LIN {X 0,Y 448.387,Z 731.206,A -85,B 0,C 180,E1 -8746.152,E2 -8746.152} C_VEL
LIN {X 0,Y 449.35,Z 719.289,A -85,B 0,C 180,E1 -8747.497,E2 -8747.497} C_VEL
LIN {X 0,Y 450.298,Z 706.862,A -85,B 0,C 180,E1 -8748.658,E2 -8748.658} C_VEL
LIN {X 0,Y 451.248,Z 693.533,A -85,B 0,C 180,E1 -8749.68,E2 -8749.68} C_VEL
LIN {X 0,Y 452.18,Z 678.745,A -85,B 0,C 180,E1 -8750.586,E2 -8750.586} C_VEL
LIN {X 0,Y 452.945,Z 663.719,A -85,B 0,C 180,E1 -8751.29,E2 -8751.29} C_VEL
LIN {X 0,Y 453.549,Z 648.187,A -85,B 0,C 180,E1 -8751.811,E2 -8751.811} C_VEL
LIN {X 0,Y 453.905,Z 632.846,A -85,B 0,C 180,E1 -8752.142,E2 -8752.142} C_VEL
LIN {X 0,Y 455.724,Z 493.743,A -85,B 0,C 180,E1 -8754.379,E2 -8754.379} C_VEL
LIN {X 0,Y 451.739,Z 464.618,A -85,B 0,C 180,E1 -8755.125,E2 -8755.125} C_VEL
LIN {X 0,Y 451.619,Z 462.28,A -85,B 0,C 180,E1 -8755.248,E2 -8755.248} C_VEL
LIN {X 0,Y 453.55,Z 429.737,A -85,B 0,C 180,E1 -8758.834,E2 -8758.834} C_VEL
LIN {X 0,Y 455.129,Z 405.936,A -85,B 0,C 180,E1 -8761.497,E2 -8761.497} C_VEL
LIN {X 0,Y 451.572,Z 392.919,A -85,B 0,C 180,E1 -8763.254,E2 -8763.254} C_VEL
LIN {X 0,Y 446.431,Z 375.769,A -85,B 0,C 180,E1 -8765.709,E2 -8765.709} C_VEL
LIN {X 0,Y 446.382,Z 375.506,A -85,B 0,C 180,E1 -8766.745,E2 -8766.745} C_VEL
LIN {X 0,Y 446.386,Z 375.51,A -85,B 0,C 180,E1 -8770.202,E2 -8770.202} C_VEL
LIN {X 0,Y 446.38,Z 375.506,A -85,B 0,C 180,E1 -8773.594,E2 -8773.594} C_VEL
LIN {X 0,Y 446.365,Z 375.494,A -85,B 0,C 180,E1 -8776.405,E2 -8776.405} C_VEL
LIN {X 0,Y 446.384,Z 375.498,A -85,B 0,C 180,E1 -8779.796,E2 -8779.796} C_VEL
LIN {X 0,Y 446.378,Z 375.492,A -85,B 0,C 180,E1 -8783.252,E2 -8783.252} C_VEL
LIN {X 0,Y 446.435,Z 375.484,A -85,B 0,C 180,E1 -8786.565,E2 -8786.565} C_VEL
LIN {X 0,Y 446.414,Z 375.501,A -85,B 0,C 180,E1 -8789.979,E2 -8789.979} C_VEL
LIN {X 0,Y 446.381,Z 375.507,A -85,B 0,C 180,E1 -8792.833,E2 -8792.833} C_VEL
LIN {X 0,Y 446.416,Z 375.492,A -85,B 0,C 180,E1 -8795.933,E2 -8795.933} C_VEL
LIN {X 0,Y 446.436,Z 375.494,A -85,B 0,C 180,E1 -8798.772,E2 -8798.772} C_VEL
LIN {X 0,Y 446.423,Z 375.497,A -85,B 0,C 180,E1 -8801.648,E2 -8801.648} C_VEL
LIN {X 0,Y 446.442,Z 375.491,A -85,B 0,C 180,E1 -8804.478,E2 -8804.478} C_VEL
LIN {X 0,Y 446.5,Z 375.489,A -85,B 0,C 180,E1 -8807.384,E2 -8807.384} C_VEL
LIN {X 0,Y 446.495,Z 375.484,A -85,B 0,C 180,E1 -8810.944,E2 -8810.944} C_VEL
LIN {X 0,Y 446.582,Z 375.478,A -85,B 0,C 180,E1 -8813.675,E2 -8813.675} C_VEL
LIN {X 0,Y 446.646,Z 375.469,A -85,B 0,C 180,E1 -8817.294,E2 -8817.294} C_VEL
LIN {X 0,Y 446.68,Z 375.466,A -85,B 0,C 180,E1 -8820,E2 -8820} C_VEL
LIN {X 0,Y 446.641,Z 375.472,A -85,B 0,C 180,E1 -8822.706,E2 -8822.706} C_VEL
LIN {X 0,Y 446.608,Z 375.47,A -85,B 0,C 180,E1 -8826.324,E2 -8826.324} C_VEL
LIN {X 0,Y 446.505,Z 375.49,A -85,B 0,C 180,E1 -8829.056,E2 -8829.056} C_VEL
LIN {X 0,Y 446.506,Z 375.484,A -85,B 0,C 180,E1 -8832.73,E2 -8832.73} C_VEL
LIN {X 0,Y 446.473,Z 375.486,A -85,B 0,C 180,E1 -8836.46,E2 -8836.46} C_VEL
LIN {X 0,Y 446.453,Z 375.494,A -85,B 0,C 180,E1 -8839.304,E2 -8839.304} C_VEL
LIN {X 0,Y 446.401,Z 375.497,A -85,B 0,C 180,E1 -8842.201,E2 -8842.201} C_VEL
LIN {X 0,Y 446.399,Z 375.496,A -85,B 0,C 180,E1 -8845.156,E2 -8845.156} C_VEL
LIN {X 0,Y 446.402,Z 375.504,A -85,B 0,C 180,E1 -8848.184,E2 -8848.184} C_VEL
LIN {X 0,Y 446.379,Z 375.507,A -85,B 0,C 180,E1 -8851.303,E2 -8851.303} C_VEL
LIN {X 0,Y 446.409,Z 375.507,A -85,B 0,C 180,E1 -8854.525,E2 -8854.525} C_VEL
LIN {X 0,Y 446.386,Z 375.486,A -85,B 0,C 180,E1 -8858.078,E2 -8858.078} C_VEL
LIN {X 0,Y 446.388,Z 375.497,A -85,B 0,C 180,E1 -8861.396,E2 -8861.396} C_VEL
LIN {X 0,Y 446.405,Z 375.504,A -85,B 0,C 180,E1 -8865.11,E2 -8865.11} C_VEL
LIN {X 0,Y 446.389,Z 375.51,A -85,B 0,C 180,E1 -8868.607,E2 -8868.607} C_VEL
LIN {X 0,Y 446.388,Z 375.506,A -85,B 0,C 180,E1 -8871.925,E2 -8871.925} C_VEL
LIN {X 0,Y 446.403,Z 375.73,A -85,B 0,C 180,E1 -8873.134,E2 -8873.134} C_VEL
LIN {X 0,Y 451.361,Z 391.214,A -85,B 0,C 180,E1 -8875.416,E2 -8875.416} C_VEL
LIN {X 0,Y 455.662,Z 406.671,A -85,B 0,C 180,E1 -8877.56,E2 -8877.56} C_VEL
LIN {X 0,Y 454.897,Z 422.239,A -85,B 0,C 180,E1 -8879.349,E2 -8879.349} C_VEL
LIN {X 0,Y 453.716,Z 445.705,A -85,B 0,C 180,E1 -8881.997,E2 -8881.997} C_VEL
LIN {X 0,Y 452.629,Z 471.656,A -85,B 0,C 180,E1 -8884.802,E2 -8884.802} C_VEL
LIN {X 0,Y 453.796,Z 479.214,A -85,B 0,C 180,E1 -8885.035,E2 -8885.035} C_VEL
LIN {X 0,Y 456.513,Z 495.836,A -85,B 0,C 180,E1 -8885.476,E2 -8885.476} C_VEL
LIN {X 0,Y 455.399,Z 574.472,A -85,B 0,C 180,E1 -8886.745,E2 -8886.745} C_VEL
LIN {X 0,Y 454.701,Z 580.317,A -85,B 0,C 180,E1 -8886.806,E2 -8886.806} C_VEL
LIN {X 0,Y 449.167,Z 599.361,A -85,B 0,C 180,E1 -8886.83,E2 -8886.83} C_VEL
LIN {X 0,Y 448.435,Z 605.208,A -85,B 0,C 180,E1 -8886.89,E2 -8886.89} C_VEL
LIN {X 0,Y 447.794,Z 641.594,A -85,B 0,C 180,E1 -8887.51,E2 -8887.51} C_VEL
LIN {X 0,Y 447.297,Z 656.597,A -85,B 0,C 180,E1 -8887.935,E2 -8887.935} C_VEL
LIN {X 0,Y 446.583,Z 670.422,A -85,B 0,C 180,E1 -8888.489,E2 -8888.489} C_VEL
LIN {X 0,Y 445.726,Z 684.345,A -85,B 0,C 180,E1 -8889.222,E2 -8889.222} C_VEL
LIN {X 0,Y 444.669,Z 698.114,A -85,B 0,C 180,E1 -8890.137,E2 -8890.137} C_VEL
LIN {X 0,Y 443.595,Z 712.023,A -85,B 0,C 180,E1 -8891.289,E2 -8891.289} C_VEL
LIN {X 0,Y 442.535,Z 724.573,A -85,B 0,C 180,E1 -8892.559,E2 -8892.559} C_VEL
LIN {X 0,Y 441.589,Z 735.099,A -85,B 0,C 180,E1 -8893.83,E2 -8893.83} C_VEL
LIN {X 0,Y 440.61,Z 746.313,A -85,B 0,C 180,E1 -8895.452,E2 -8895.452} C_VEL
LIN {X 0,Y 439.871,Z 755.606,A -85,B 0,C 180,E1 -8897.076,E2 -8897.076} C_VEL
LIN {X 0,Y 439.437,Z 762.344,A -85,B 0,C 180,E1 -8898.47,E2 -8898.47} C_VEL
LIN {X 0,Y 438.855,Z 769.757,A -85,B 0,C 180,E1 -8900.321,E2 -8900.321} C_VEL
LIN {X 0,Y 438.543,Z 775.645,A -85,B 0,C 180,E1 -8902.172,E2 -8902.172} C_VEL
LIN {X 0,Y 438.365,Z 779.494,A -85,B 0,C 180,E1 -8903.723,E2 -8903.723} C_VEL
LIN {X 0,Y 438.3,Z 782.66,A -85,B 0,C 180,E1 -8905.403,E2 -8905.403} C_VEL
LIN {X 0,Y 438.286,Z 785.001,A -85,B 0,C 180,E1 -8907.244,E2 -8907.244} C_VEL
LIN {X 0,Y 438.227,Z 786.195,A -85,B 0,C 180,E1 -8909.083,E2 -8909.083} C_VEL
LIN {X 0,Y 438.228,Z 786.212,A -85,B 0,C 180,E1 -8910.92,E2 -8910.92} C_VEL
LIN {X 0,Y 438.287,Z 785.081,A -85,B 0,C 180,E1 -8912.759,E2 -8912.759} C_VEL
LIN {X 0,Y 438.3,Z 782.802,A -85,B 0,C 180,E1 -8914.6,E2 -8914.6} C_VEL
LIN {X 0,Y 438.448,Z 779.319,A -85,B 0,C 180,E1 -8916.444,E2 -8916.444} C_VEL
LIN {X 0,Y 438.614,Z 774.553,A -85,B 0,C 180,E1 -8918.293,E2 -8918.293} C_VEL
LIN {X 0,Y 438.915,Z 768.383,A -85,B 0,C 180,E1 -8920.146,E2 -8920.146} C_VEL
LIN {X 0,Y 439.484,Z 761.721,A -85,B 0,C 180,E1 -8921.766,E2 -8921.766} C_VEL
LIN {X 0,Y 439.987,Z 753.641,A -85,B 0,C 180,E1 -8923.393,E2 -8923.393} C_VEL
LIN {X 0,Y 440.822,Z 743.941,A -85,B 0,C 180,E1 -8925.016,E2 -8925.016} C_VEL
LIN {X 0,Y 441.873,Z 732.205,A -85,B 0,C 180,E1 -8926.637,E2 -8926.637} C_VEL
LIN {X 0,Y 442.903,Z 720.026,A -85,B 0,C 180,E1 -8928.025,E2 -8928.025} C_VEL
LIN {X 0,Y 443.962,Z 707.857,A -85,B 0,C 180,E1 -8929.178,E2 -8929.178} C_VEL
LIN {X 0,Y 444.962,Z 694.601,A -85,B 0,C 180,E1 -8930.214,E2 -8930.214} C_VEL
LIN {X 0,Y 445.986,Z 680.954,A -85,B 0,C 180,E1 -8931.07,E2 -8931.07} C_VEL
LIN {X 0,Y 446.838,Z 665.339,A -85,B 0,C 180,E1 -8931.83,E2 -8931.83} C_VEL
LIN {X 0,Y 447.576,Z 650.475,A -85,B 0,C 180,E1 -8932.353,E2 -8932.353} C_VEL
LIN {X 0,Y 447.983,Z 636.081,A -85,B 0,C 180,E1 -8932.696,E2 -8932.696} C_VEL
LIN {X 0,Y 450.045,Z 497.422,A -85,B 0,C 180,E1 -8934.965,E2 -8934.965} C_VEL
LIN {X 0,Y 446.021,Z 472.043,A -85,B 0,C 180,E1 -8935.664,E2 -8935.664} C_VEL
LIN {X 0,Y 446.629,Z 455.684,A -85,B 0,C 180,E1 -8937.406,E2 -8937.406} C_VEL
LIN {X 0,Y 447.911,Z 431.433,A -85,B 0,C 180,E1 -8940.14,E2 -8940.14} C_VEL
LIN {X 0,Y 449.103,Z 409.391,A -85,B 0,C 180,E1 -8942.677,E2 -8942.677} C_VEL
LIN {X 0,Y 445.361,Z 395.604,A -85,B 0,C 180,E1 -8944.619,E2 -8944.619} C_VEL
LIN {X 0,Y 440.841,Z 381.251,A -85,B 0,C 180,E1 -8946.713,E2 -8946.713} C_VEL
LIN {X 0,Y 439.357,Z 376.547,A -85,B 0,C 180,E1 -8947.472,E2 -8947.472} C_VEL
LIN {X 0,Y 439.35,Z 376.378,A -85,B 0,C 180,E1 -8949.841,E2 -8949.841} C_VEL
LIN {X 0,Y 439.332,Z 376.374,A -85,B 0,C 180,E1 -8952.62,E2 -8952.62} C_VEL
LIN {X 0,Y 439.37,Z 376.367,A -85,B 0,C 180,E1 -8955.267,E2 -8955.267} C_VEL
LIN {X 0,Y 439.362,Z 376.374,A -85,B 0,C 180,E1 -8958.749,E2 -8958.749} C_VEL
LIN {X 0,Y 439.356,Z 376.381,A -85,B 0,C 180,E1 -8961.612,E2 -8961.612} C_VEL
LIN {X 0,Y 439.392,Z 376.357,A -85,B 0,C 180,E1 -8964.843,E2 -8964.843} C_VEL
LIN {X 0,Y 439.35,Z 376.381,A -85,B 0,C 180,E1 -8968.138,E2 -8968.138} C_VEL
LIN {X 0,Y 439.384,Z 376.381,A -85,B 0,C 180,E1 -8971.324,E2 -8971.324} C_VEL
LIN {X 0,Y 439.358,Z 376.382,A -85,B 0,C 180,E1 -8974.412,E2 -8974.412} C_VEL
LIN {X 0,Y 439.455,Z 376.495,A -85,B 0,C 180,E1 -8976.558,E2 -8976.558} C_VEL
LIN {X 0,Y 441.167,Z 384.3,A -85,B 0,C 180,E1 -8978.12,E2 -8978.12} C_VEL
LIN {X 0,Y 443.676,Z 391.102,A -85,B 0,C 180,E1 -8978.416,E2 -8978.416} C_VEL
LIN {X 0,Y 446.444,Z 399.4,A -85,B 0,C 180,E1 -8978.714,E2 -8978.714} C_VEL
LIN {X 0,Y 446.853,Z 402.358,A -85,B 0,C 180,E1 -8978.793,E2 -8978.793} C_VEL
LIN {X 0,Y 444.571,Z 525.307,A -85,B 0,C 180,E1 -8981.15,E2 -8981.15} C_VEL
LIN {X 0,Y 444.383,Z 540.563,A -85,B 0,C 180,E1 -8981.643,E2 -8981.643} C_VEL
LIN {X 0,Y 443.976,Z 555.135,A -85,B 0,C 180,E1 -8982.306,E2 -8982.306} C_VEL
LIN {X 0,Y 443.458,Z 568.001,A -85,B 0,C 180,E1 -8983.069,E2 -8983.069} C_VEL
LIN {X 0,Y 442.975,Z 579.027,A -85,B 0,C 180,E1 -8983.88,E2 -8983.88} C_VEL
LIN {X 0,Y 442.318,Z 591.98,A -85,B 0,C 180,E1 -8985.037,E2 -8985.037} C_VEL
LIN {X 0,Y 441.734,Z 602.587,A -85,B 0,C 180,E1 -8986.193,E2 -8986.193} C_VEL
LIN {X 0,Y 441.248,Z 611.484,A -85,B 0,C 180,E1 -8987.349,E2 -8987.349} C_VEL
LIN {X 0,Y 440.72,Z 620.489,A -85,B 0,C 180,E1 -8988.735,E2 -8988.735} C_VEL
LIN {X 0,Y 440.285,Z 629.099,A -85,B 0,C 180,E1 -8990.351,E2 -8990.351} C_VEL
LIN {X 0,Y 439.978,Z 635.137,A -85,B 0,C 180,E1 -8991.734,E2 -8991.734} C_VEL
LIN {X 0,Y 439.772,Z 640.064,A -85,B 0,C 180,E1 -8993.116,E2 -8993.116} C_VEL
LIN {X 0,Y 439.509,Z 645.241,A -85,B 0,C 180,E1 -8994.954,E2 -8994.954} C_VEL
LIN {X 0,Y 439.266,Z 648.069,A -85,B 0,C 180,E1 -8996.331,E2 -8996.331} C_VEL
LIN {X 0,Y 439.371,Z 649.493,A -85,B 0,C 180,E1 -8997.249,E2 -8997.249} C_VEL
LIN {X 0,Y 439.323,Z 651.335,A -85,B 0,C 180,E1 -8999.083,E2 -8999.083} C_VEL
LIN {X 0,Y 439.336,Z 651.805,A -85,B 0,C 180,E1 -9000.916,E2 -9000.916} C_VEL
LIN {X 0,Y 439.532,Z 650.857,A -85,B 0,C 180,E1 -9002.749,E2 -9002.749} C_VEL
LIN {X 0,Y 439.63,Z 648.519,A -85,B 0,C 180,E1 -9004.585,E2 -9004.585} C_VEL
LIN {X 0,Y 440.034,Z 644.689,A -85,B 0,C 180,E1 -9006.419,E2 -9006.419} C_VEL
LIN {X 0,Y 440.418,Z 640.115,A -85,B 0,C 180,E1 -9008.007,E2 -9008.007} C_VEL
LIN {X 0,Y 440.862,Z 634.054,A -85,B 0,C 180,E1 -9009.636,E2 -9009.636} C_VEL
LIN {X 0,Y 441.488,Z 626.483,A -85,B 0,C 180,E1 -9011.245,E2 -9011.245} C_VEL
LIN {X 0,Y 442.092,Z 618.506,A -85,B 0,C 180,E1 -9012.626,E2 -9012.626} C_VEL
LIN {X 0,Y 442.822,Z 608.572,A -85,B 0,C 180,E1 -9014.049,E2 -9014.049} C_VEL
LIN {X 0,Y 443.565,Z 598.173,A -85,B 0,C 180,E1 -9015.272,E2 -9015.272} C_VEL
LIN {X 0,Y 444.272,Z 586.188,A -85,B 0,C 180,E1 -9016.425,E2 -9016.425} C_VEL
LIN {X 0,Y 444.837,Z 574.421,A -85,B 0,C 180,E1 -9017.35,E2 -9017.35} C_VEL
LIN {X 0,Y 445.484,Z 560.513,A -85,B 0,C 180,E1 -9018.214,E2 -9018.214} C_VEL
LIN {X 0,Y 445.951,Z 547.604,A -85,B 0,C 180,E1 -9018.836,E2 -9018.836} C_VEL
LIN {X 0,Y 446.202,Z 533.444,A -85,B 0,C 180,E1 -9019.345,E2 -9019.345} C_VEL
LIN {X 0,Y 447.324,Z 488.713,A -85,B 0,C 180,E1 -9020.371,E2 -9020.371} C_VEL
LIN {X 0,Y 450.617,Z 407.034,A -85,B 0,C 180,E1 -9022.286,E2 -9022.286} C_VEL
LIN {X 0,Y 449.747,Z 404.596,A -85,B 0,C 180,E1 -9022.421,E2 -9022.421} C_VEL
LIN {X 0,Y 444.925,Z 395.422,A -85,B 0,C 180,E1 -9023.126,E2 -9023.126} C_VEL
LIN {X 0,Y 442.843,Z 387.302,A -85,B 0,C 180,E1 -9025.372,E2 -9025.372} C_VEL
LIN {X 0,Y 440.221,Z 378.808,A -85,B 0,C 180,E1 -9028.051,E2 -9028.051} C_VEL
LIN {X 0,Y 439.434,Z 376.439,A -85,B 0,C 180,E1 -9028.934,E2 -9028.934} C_VEL
LIN {X 0,Y 439.375,Z 376.382,A -85,B 0,C 180,E1 -9032.03,E2 -9032.03} C_VEL
LIN {X 0,Y 439.398,Z 376.378,A -85,B 0,C 180,E1 -9035.339,E2 -9035.339} C_VEL
LIN {X 0,Y 439.373,Z 376.382,A -85,B 0,C 180,E1 -9038.596,E2 -9038.596} C_VEL
LIN {X 0,Y 439.385,Z 376.379,A -85,B 0,C 180,E1 -9041.255,E2 -9041.255} C_VEL
LIN {X 0,Y 439.402,Z 376.379,A -85,B 0,C 180,E1 -9044.729,E2 -9044.729} C_VEL
LIN {X 0,Y 439.355,Z 376.384,A -85,B 0,C 180,E1 -9047.79,E2 -9047.79} C_VEL
LIN {X 0,Y 439.362,Z 376.384,A -85,B 0,C 180,E1 -9050.219,E2 -9050.219} C_VEL
LIN {X 0,Y 439.381,Z 376.649,A -85,B 0,C 180,E1 -9051.568,E2 -9051.568} C_VEL
LIN {X 0,Y 442.526,Z 384.848,A -85,B 0,C 180,E1 -9053.627,E2 -9053.627} C_VEL
LIN {X 0,Y 445.548,Z 393.892,A -85,B 0,C 180,E1 -9055.505,E2 -9055.505} C_VEL
LIN {X 0,Y 448.186,Z 403.614,A -85,B 0,C 180,E1 -9057.248,E2 -9057.248} C_VEL
LIN {X 0,Y 449.288,Z 408.646,A -85,B 0,C 180,E1 -9058.059,E2 -9058.059} C_VEL
LIN {X 0,Y 446.963,Z 431.712,A -85,B 0,C 180,E1 -9060.955,E2 -9060.955} C_VEL
LIN {X 0,Y 444.894,Z 457.945,A -85,B 0,C 180,E1 -9064.059,E2 -9064.059} C_VEL
LIN {X 0,Y 447.037,Z 473.427,A -85,B 0,C 180,E1 -9064.62,E2 -9064.62} C_VEL
LIN {X 0,Y 449.286,Z 495.995,A -85,B 0,C 180,E1 -9065.282,E2 -9065.282} C_VEL
LIN {X 0,Y 447.324,Z 637.604,A -85,B 0,C 180,E1 -9067.603,E2 -9067.603} C_VEL
LIN {X 0,Y 446.884,Z 652.57,A -85,B 0,C 180,E1 -9067.982,E2 -9067.982} C_VEL
LIN {X 0,Y 446.231,Z 666.921,A -85,B 0,C 180,E1 -9068.516,E2 -9068.516} C_VEL
LIN {X 0,Y 445.422,Z 680.779,A -85,B 0,C 180,E1 -9069.205,E2 -9069.205} C_VEL
LIN {X 0,Y 444.622,Z 693.569,A -85,B 0,C 180,E1 -9070.011,E2 -9070.011} C_VEL
LIN {X 0,Y 443.558,Z 706.88,A -85,B 0,C 180,E1 -9071.044,E2 -9071.044} C_VEL
LIN {X 0,Y 442.586,Z 719.085,A -85,B 0,C 180,E1 -9072.2,E2 -9072.2} C_VEL
LIN {X 0,Y 441.55,Z 731.221,A -85,B 0,C 180,E1 -9073.588,E2 -9073.588} C_VEL
LIN {X 0,Y 440.752,Z 741.388,A -85,B 0,C 180,E1 -9074.981,E2 -9074.981} C_VEL
LIN {X 0,Y 439.945,Z 751.301,A -85,B 0,C 180,E1 -9076.605,E2 -9076.605} C_VEL
LIN {X 0,Y 439.437,Z 759.517,A -85,B 0,C 180,E1 -9078.233,E2 -9078.233} C_VEL
LIN {X 0,Y 438.912,Z 766.306,A -85,B 0,C 180,E1 -9079.854,E2 -9079.854} C_VEL
LIN {X 0,Y 438.637,Z 772.585,A -85,B 0,C 180,E1 -9081.708,E2 -9081.708} C_VEL
LIN {X 0,Y 438.505,Z 777.436,A -85,B 0,C 180,E1 -9083.557,E2 -9083.557} C_VEL
LIN {X 0,Y 438.376,Z 780.987,A -85,B 0,C 180,E1 -9085.401,E2 -9085.401} C_VEL
LIN {X 0,Y 438.406,Z 783.32,A -85,B 0,C 180,E1 -9087.242,E2 -9087.242} C_VEL
LIN {X 0,Y 438.297,Z 784.492,A -85,B 0,C 180,E1 -9089.08,E2 -9089.08} C_VEL
LIN {X 0,Y 438.296,Z 784.491,A -85,B 0,C 180,E1 -9090.917,E2 -9090.917} C_VEL
LIN {X 0,Y 438.41,Z 783.317,A -85,B 0,C 180,E1 -9092.755,E2 -9092.755} C_VEL
LIN {X 0,Y 438.36,Z 780.985,A -85,B 0,C 180,E1 -9094.596,E2 -9094.596} C_VEL
LIN {X 0,Y 438.444,Z 777.441,A -85,B 0,C 180,E1 -9096.441,E2 -9096.441} C_VEL
LIN {X 0,Y 438.627,Z 772.592,A -85,B 0,C 180,E1 -9098.29,E2 -9098.29} C_VEL
LIN {X 0,Y 438.908,Z 766.306,A -85,B 0,C 180,E1 -9100.143,E2 -9100.143} C_VEL
LIN {X 0,Y 439.413,Z 759.516,A -85,B 0,C 180,E1 -9101.765,E2 -9101.765} C_VEL
LIN {X 0,Y 439.938,Z 751.305,A -85,B 0,C 180,E1 -9103.392,E2 -9103.392} C_VEL
LIN {X 0,Y 440.704,Z 741.393,A -85,B 0,C 180,E1 -9105.017,E2 -9105.017} C_VEL
LIN {X 0,Y 441.514,Z 731.227,A -85,B 0,C 180,E1 -9106.41,E2 -9106.41} C_VEL
LIN {X 0,Y 442.548,Z 719.312,A -85,B 0,C 180,E1 -9107.775,E2 -9107.775} C_VEL
LIN {X 0,Y 443.531,Z 706.888,A -85,B 0,C 180,E1 -9108.954,E2 -9108.954} C_VEL
LIN {X 0,Y 444.543,Z 693.563,A -85,B 0,C 180,E1 -9109.99,E2 -9109.99} C_VEL
LIN {X 0,Y 445.531,Z 678.784,A -85,B 0,C 180,E1 -9110.908,E2 -9110.908} C_VEL
LIN {X 0,Y 446.364,Z 663.55,A -85,B 0,C 180,E1 -9111.629,E2 -9111.629} C_VEL
LIN {X 0,Y 446.966,Z 648.311,A -85,B 0,C 180,E1 -9112.148,E2 -9112.148} C_VEL
LIN {X 0,Y 447.338,Z 632.974,A -85,B 0,C 180,E1 -9112.484,E2 -9112.484} C_VEL
LIN {X 0,Y 449.286,Z 494.748,A -85,B 0,C 180,E1 -9114.736,E2 -9114.736} C_VEL
LIN {X 0,Y 445.192,Z 464.342,A -85,B 0,C 180,E1 -9115.535,E2 -9115.535} C_VEL
LIN {X 0,Y 444.904,Z 460.81,A -85,B 0,C 180,E1 -9115.713,E2 -9115.713} C_VEL
LIN {X 0,Y 446.946,Z 428.713,A -85,B 0,C 180,E1 -9119.301,E2 -9119.301} C_VEL
LIN {X 0,Y 448.334,Z 408.594,A -85,B 0,C 180,E1 -9121.589,E2 -9121.589} C_VEL
LIN {X 0,Y 448.031,Z 406.17,A -85,B 0,C 180,E1 -9121.894,E2 -9121.894} C_VEL
LIN {X 0,Y 442.305,Z 386.339,A -85,B 0,C 180,E1 -9124.662,E2 -9124.662} C_VEL
LIN {X 0,Y 439.404,Z 376.558,A -85,B 0,C 180,E1 -9126.124,E2 -9126.124} C_VEL
LIN {X 0,Y 439.348,Z 376.384,A -85,B 0,C 180,E1 -9129.779,E2 -9129.779} C_VEL
LIN {X 0,Y 439.331,Z 376.387,A -85,B 0,C 180,E1 -9132.62,E2 -9132.62} C_VEL
LIN {X 0,Y 439.36,Z 376.379,A -85,B 0,C 180,E1 -9135.266,E2 -9135.266} C_VEL
LIN {X 0,Y 439.34,Z 376.368,A -85,B 0,C 180,E1 -9139.015,E2 -9139.015} C_VEL
LIN {X 0,Y 439.342,Z 376.382,A -85,B 0,C 180,E1 -9141.61,E2 -9141.61} C_VEL
LIN {X 0,Y 439.377,Z 376.345,A -85,B 0,C 180,E1 -9144.842,E2 -9144.842} C_VEL
LIN {X 0,Y 439.355,Z 376.38,A -85,B 0,C 180,E1 -9148.138,E2 -9148.138} C_VEL
LIN {X 0,Y 439.385,Z 376.37,A -85,B 0,C 180,E1 -9151.605,E2 -9151.605} C_VEL
LIN {X 0,Y 439.352,Z 376.376,A -85,B 0,C 180,E1 -9154.412,E2 -9154.412} C_VEL
LIN {X 0,Y 439.346,Z 376.38,A -85,B 0,C 180,E1 -9157.424,E2 -9157.424} C_VEL
LIN {X 0,Y 439.425,Z 376.366,A -85,B 0,C 180,E1 -9160.663,E2 -9160.663} C_VEL
LIN {X 0,Y 439.402,Z 376.371,A -85,B 0,C 180,E1 -9164.222,E2 -9164.222} C_VEL
LIN {X 0,Y 439.469,Z 376.365,A -85,B 0,C 180,E1 -9167.285,E2 -9167.285} C_VEL
LIN {X 0,Y 439.461,Z 376.359,A -85,B 0,C 180,E1 -9170.798,E2 -9170.798} C_VEL
LIN {X 0,Y 439.533,Z 376.356,A -85,B 0,C 180,E1 -9173.574,E2 -9173.574} C_VEL
LIN {X 0,Y 439.394,Z 376.362,A -85,B 0,C 180,E1 -9175.413,E2 -9175.413} C_VEL
LIN {X 0,Y 439.614,Z 376.348,A -85,B 0,C 180,E1 -9178.168,E2 -9178.168} C_VEL
LIN {X 0,Y 439.579,Z 376.342,A -85,B 0,C 180,E1 -9180.916,E2 -9180.916} C_VEL
LIN {X 0,Y 439.593,Z 376.35,A -85,B 0,C 180,E1 -9182.749,E2 -9182.749} C_VEL
LIN {X 0,Y 439.579,Z 376.344,A -85,B 0,C 180,E1 -9186.426,E2 -9186.426} C_VEL
LIN {X 0,Y 439.469,Z 376.365,A -85,B 0,C 180,E1 -9189.202,E2 -9189.202} C_VEL
LIN {X 0,Y 439.45,Z 376.366,A -85,B 0,C 180,E1 -9192.938,E2 -9192.938} C_VEL
LIN {X 0,Y 439.431,Z 376.363,A -85,B 0,C 180,E1 -9196.349,E2 -9196.349} C_VEL
LIN {X 0,Y 439.387,Z 376.373,A -85,B 0,C 180,E1 -9199.627,E2 -9199.627} C_VEL
LIN {X 0,Y 439.347,Z 376.38,A -85,B 0,C 180,E1 -9202.577,E2 -9202.577} C_VEL
LIN {X 0,Y 439.339,Z 376.375,A -85,B 0,C 180,E1 -9205.589,E2 -9205.589} C_VEL
LIN {X 0,Y 439.366,Z 376.377,A -85,B 0,C 180,E1 -9208.677,E2 -9208.677} C_VEL
LIN {X 0,Y 439.338,Z 376.383,A -85,B 0,C 180,E1 -9212.028,E2 -9212.028} C_VEL
LIN {X 0,Y 439.377,Z 376.376,A -85,B 0,C 180,E1 -9215.341,E2 -9215.341} C_VEL
LIN {X 0,Y 439.343,Z 376.368,A -85,B 0,C 180,E1 -9218.599,E2 -9218.599} C_VEL
LIN {X 0,Y 439.335,Z 376.368,A -85,B 0,C 180,E1 -9222.212,E2 -9222.212} C_VEL
LIN {X 0,Y 439.36,Z 376.38,A -85,B 0,C 180,E1 -9225.268,E2 -9225.268} C_VEL
LIN {X 0,Y 439.343,Z 376.382,A -85,B 0,C 180,E1 -9229.018,E2 -9229.018} C_VEL
LIN {X 0,Y 439.358,Z 376.468,A -85,B 0,C 180,E1 -9232.603,E2 -9232.603} C_VEL
LIN {X 0,Y 439.456,Z 377.028,A -85,B 0,C 180,E1 -9232.749,E2 -9232.749} C_VEL
LIN {X 0,Y 444.405,Z 392.208,A -85,B 0,C 180,E1 -9235.001,E2 -9235.001} C_VEL
LIN {X 0,Y 449.012,Z 408.606,A -85,B 0,C 180,E1 -9237.319,E2 -9237.319} C_VEL
LIN {X 0,Y 448.891,Z 414.13,A -85,B 0,C 180,E1 -9237.972,E2 -9237.972} C_VEL
LIN {X 0,Y 447.377,Z 441.599,A -85,B 0,C 180,E1 -9241.117,E2 -9241.117} C_VEL
LIN {X 0,Y 446.117,Z 468.485,A -85,B 0,C 180,E1 -9244.079,E2 -9244.079} C_VEL
LIN {X 0,Y 445.995,Z 472.091,A -85,B 0,C 180,E1 -9244.432,E2 -9244.432} C_VEL
LIN {X 0,Y 450.042,Z 496.761,A -85,B 0,C 180,E1 -9245.117,E2 -9245.117} C_VEL
LIN {X 0,Y 448.435,Z 605.208,A -85,B 0,C 180,E1 -9246.89,E2 -9246.89} C_VEL
LIN {X 0,Y 447.707,Z 611.054,A -85,B 0,C 180,E1 -9246.95,E2 -9246.95} C_VEL
LIN {X 0,Y 442.162,Z 630.092,A -85,B 0,C 180,E1 -9246.976,E2 -9246.976} C_VEL
LIN {X 0,Y 441.423,Z 635.933,A -85,B 0,C 180,E1 -9247.041,E2 -9247.041} C_VEL
LIN {X 0,Y 440.956,Z 651.478,A -85,B 0,C 180,E1 -9247.42,E2 -9247.42} C_VEL
LIN {X 0,Y 440.244,Z 666.161,A -85,B 0,C 180,E1 -9247.957,E2 -9247.957} C_VEL
LIN {X 0,Y 439.39,Z 680.397,A -85,B 0,C 180,E1 -9248.663,E2 -9248.663} C_VEL
LIN {X 0,Y 438.264,Z 694.991,A -85,B 0,C 180,E1 -9249.589,E2 -9249.589} C_VEL
LIN {X 0,Y 437.171,Z 708.187,A -85,B 0,C 180,E1 -9250.638,E2 -9250.638} C_VEL
LIN {X 0,Y 436.059,Z 720.812,A -85,B 0,C 180,E1 -9251.861,E2 -9251.861} C_VEL
LIN {X 0,Y 435.077,Z 731.467,A -85,B 0,C 180,E1 -9253.098,E2 -9253.098} C_VEL
LIN {X 0,Y 434.1,Z 741.757,A -85,B 0,C 180,E1 -9254.508,E2 -9254.508} C_VEL
LIN {X 0,Y 433.186,Z 751.824,A -85,B 0,C 180,E1 -9256.156,E2 -9256.156} C_VEL
LIN {X 0,Y 432.525,Z 760.184,A -85,B 0,C 180,E1 -9257.807,E2 -9257.807} C_VEL
LIN {X 0,Y 432.062,Z 766.238,A -85,B 0,C 180,E1 -9259.22,E2 -9259.22} C_VEL
LIN {X 0,Y 431.624,Z 772.867,A -85,B 0,C 180,E1 -9261.103,E2 -9261.103} C_VEL
LIN {X 0,Y 431.376,Z 778.053,A -85,B 0,C 180,E1 -9262.983,E2 -9262.983} C_VEL
LIN {X 0,Y 431.247,Z 781.03,A -85,B 0,C 180,E1 -9264.39,E2 -9264.39} C_VEL
LIN {X 0,Y 431.148,Z 783.963,A -85,B 0,C 180,E1 -9266.263,E2 -9266.263} C_VEL
LIN {X 0,Y 431.194,Z 785.726,A -85,B 0,C 180,E1 -9268.133,E2 -9268.133} C_VEL
LIN {X 0,Y 431.12,Z 786.339,A -85,B 0,C 180,E1 -9270.001,E2 -9270.001} C_VEL
LIN {X 0,Y 431.195,Z 785.774,A -85,B 0,C 180,E1 -9271.869,E2 -9271.869} C_VEL
LIN {X 0,Y 431.149,Z 784.073,A -85,B 0,C 180,E1 -9273.74,E2 -9273.74} C_VEL
LIN {X 0,Y 431.257,Z 781.2,A -85,B 0,C 180,E1 -9275.613,E2 -9275.613} C_VEL
LIN {X 0,Y 431.42,Z 777.086,A -85,B 0,C 180,E1 -9277.49,E2 -9277.49} C_VEL
LIN {X 0,Y 431.694,Z 771.636,A -85,B 0,C 180,E1 -9279.371,E2 -9279.371} C_VEL
LIN {X 0,Y 432.234,Z 764.698,A -85,B 0,C 180,E1 -9281.253,E2 -9281.253} C_VEL
LIN {X 0,Y 432.778,Z 756.757,A -85,B 0,C 180,E1 -9283.003,E2 -9283.003} C_VEL
LIN {X 0,Y 433.519,Z 748.303,A -85,B 0,C 180,E1 -9284.554,E2 -9284.554} C_VEL
LIN {X 0,Y 434.508,Z 737.484,A -85,B 0,C 180,E1 -9286.203,E2 -9286.203} C_VEL
LIN {X 0,Y 435.598,Z 725.65,A -85,B 0,C 180,E1 -9287.694,E2 -9287.694} C_VEL
LIN {X 0,Y 436.666,Z 714.188,A -85,B 0,C 180,E1 -9288.901,E2 -9288.901} C_VEL
LIN {X 0,Y 437.824,Z 700.767,A -85,B 0,C 180,E1 -9290.068,E2 -9290.068} C_VEL
LIN {X 0,Y 438.839,Z 687.652,A -85,B 0,C 180,E1 -9290.999,E2 -9290.999} C_VEL
LIN {X 0,Y 439.844,Z 673.529,A -85,B 0,C 180,E1 -9291.794,E2 -9291.794} C_VEL
LIN {X 0,Y 440.582,Z 658.789,A -85,B 0,C 180,E1 -9292.431,E2 -9292.431} C_VEL
LIN {X 0,Y 441.203,Z 644.049,A -85,B 0,C 180,E1 -9292.879,E2 -9292.879} C_VEL
LIN {X 0,Y 441.632,Z 621.84,A -85,B 0,C 180,E1 -9293.289,E2 -9293.289} C_VEL
LIN {X 0,Y 443.582,Z 498.768,A -85,B 0,C 180,E1 -9295.328,E2 -9295.328} C_VEL
LIN {X 0,Y 442.11,Z 488.085,A -85,B 0,C 180,E1 -9295.606,E2 -9295.606} C_VEL
LIN {X 0,Y 439.397,Z 471.699,A -85,B 0,C 180,E1 -9296.096,E2 -9296.096} C_VEL
LIN {X 0,Y 440.376,Z 450.137,A -85,B 0,C 180,E1 -9298.446,E2 -9298.446} C_VEL
LIN {X 0,Y 441.953,Z 422.246,A -85,B 0,C 180,E1 -9301.654,E2 -9301.654} C_VEL
LIN {X 0,Y 442.58,Z 412.244,A -85,B 0,C 180,E1 -9302.812,E2 -9302.812} C_VEL
LIN {X 0,Y 439.935,Z 401.732,A -85,B 0,C 180,E1 -9304.297,E2 -9304.297} C_VEL
LIN {X 0,Y 434.864,Z 385.277,A -85,B 0,C 180,E1 -9306.726,E2 -9306.726} C_VEL
LIN {X 0,Y 432.36,Z 377.5,A -85,B 0,C 180,E1 -9307.935,E2 -9307.935} C_VEL
LIN {X 0,Y 432.291,Z 377.262,A -85,B 0,C 180,E1 -9310.172,E2 -9310.172} C_VEL
LIN {X 0,Y 432.285,Z 377.257,A -85,B 0,C 180,E1 -9313.066,E2 -9313.066} C_VEL
LIN {X 0,Y 432.314,Z 377.244,A -85,B 0,C 180,E1 -9315.669,E2 -9315.669} C_VEL
LIN {X 0,Y 432.308,Z 377.259,A -85,B 0,C 180,E1 -9318.403,E2 -9318.403} C_VEL
LIN {X 0,Y 432.322,Z 377.258,A -85,B 0,C 180,E1 -9321.848,E2 -9321.848} C_VEL
LIN {X 0,Y 432.327,Z 377.235,A -85,B 0,C 180,E1 -9325.322,E2 -9325.322} C_VEL
LIN {X 0,Y 432.306,Z 377.26,A -85,B 0,C 180,E1 -9328.653,E2 -9328.653} C_VEL
LIN {X 0,Y 432.318,Z 377.258,A -85,B 0,C 180,E1 -9331.872,E2 -9331.872} C_VEL
LIN {X 0,Y 432.352,Z 377.256,A -85,B 0,C 180,E1 -9335.548,E2 -9335.548} C_VEL
LIN {X 0,Y 432.425,Z 377.501,A -85,B 0,C 180,E1 -9336.313,E2 -9336.313} C_VEL
LIN {X 0,Y 434.086,Z 385.052,A -85,B 0,C 180,E1 -9337.811,E2 -9337.811} C_VEL
LIN {X 0,Y 439.819,Z 400.86,A -85,B 0,C 180,E1 -9338.437,E2 -9338.437} C_VEL
LIN {X 0,Y 440.104,Z 403.823,A -85,B 0,C 180,E1 -9338.512,E2 -9338.512} C_VEL
LIN {X 0,Y 437.761,Z 525.926,A -85,B 0,C 180,E1 -9340.907,E2 -9340.907} C_VEL
LIN {X 0,Y 437.559,Z 540.994,A -85,B 0,C 180,E1 -9341.399,E2 -9341.399} C_VEL
LIN {X 0,Y 437.152,Z 555.016,A -85,B 0,C 180,E1 -9342.039,E2 -9342.039} C_VEL
LIN {X 0,Y 436.647,Z 567.809,A -85,B 0,C 180,E1 -9342.797,E2 -9342.797} C_VEL
LIN {X 0,Y 436.11,Z 579.041,A -85,B 0,C 180,E1 -9343.619,E2 -9343.619} C_VEL
LIN {X 0,Y 435.51,Z 590.946,A -85,B 0,C 180,E1 -9344.677,E2 -9344.677} C_VEL
LIN {X 0,Y 434.835,Z 602.907,A -85,B 0,C 180,E1 -9345.969,E2 -9345.969} C_VEL
LIN {X 0,Y 434.33,Z 611.921,A -85,B 0,C 180,E1 -9347.144,E2 -9347.144} C_VEL
LIN {X 0,Y 433.77,Z 621.034,A -85,B 0,C 180,E1 -9348.552,E2 -9348.552} C_VEL
LIN {X 0,Y 433.304,Z 629.768,A -85,B 0,C 180,E1 -9350.194,E2 -9350.194} C_VEL
LIN {X 0,Y 432.993,Z 635.864,A -85,B 0,C 180,E1 -9351.6,E2 -9351.6} C_VEL
LIN {X 0,Y 432.779,Z 640.869,A -85,B 0,C 180,E1 -9353.004,E2 -9353.004} C_VEL
LIN {X 0,Y 432.508,Z 646.117,A -85,B 0,C 180,E1 -9354.872,E2 -9354.872} C_VEL
LIN {X 0,Y 432.242,Z 649.012,A -85,B 0,C 180,E1 -9356.271,E2 -9356.271} C_VEL
LIN {X 0,Y 432.352,Z 650.466,A -85,B 0,C 180,E1 -9357.205,E2 -9357.205} C_VEL
LIN {X 0,Y 432.303,Z 652.361,A -85,B 0,C 180,E1 -9359.068,E2 -9359.068} C_VEL
LIN {X 0,Y 432.321,Z 652.886,A -85,B 0,C 180,E1 -9360.931,E2 -9360.931} C_VEL
LIN {X 0,Y 432.536,Z 652.003,A -85,B 0,C 180,E1 -9362.794,E2 -9362.794} C_VEL
LIN {X 0,Y 432.673,Z 649.717,A -85,B 0,C 180,E1 -9364.658,E2 -9364.658} C_VEL
LIN {X 0,Y 432.971,Z 647.027,A -85,B 0,C 180,E1 -9366.056,E2 -9366.056} C_VEL
LIN {X 0,Y 433.337,Z 643.441,A -85,B 0,C 180,E1 -9367.455,E2 -9367.455} C_VEL
LIN {X 0,Y 433.766,Z 638.418,A -85,B 0,C 180,E1 -9368.994,E2 -9368.994} C_VEL
LIN {X 0,Y 434.377,Z 631.254,A -85,B 0,C 180,E1 -9370.723,E2 -9370.723} C_VEL
LIN {X 0,Y 434.961,Z 624.079,A -85,B 0,C 180,E1 -9372.125,E2 -9372.125} C_VEL
LIN {X 0,Y 435.738,Z 615.374,A -85,B 0,C 180,E1 -9373.525,E2 -9373.525} C_VEL
LIN {X 0,Y 436.445,Z 606.166,A -85,B 0,C 180,E1 -9374.758,E2 -9374.758} C_VEL
LIN {X 0,Y 437.202,Z 595.199,A -85,B 0,C 180,E1 -9375.979,E2 -9375.979} C_VEL
LIN {X 0,Y 437.938,Z 582.323,A -85,B 0,C 180,E1 -9377.15,E2 -9377.15} C_VEL
LIN {X 0,Y 438.585,Z 571.229,A -85,B 0,C 180,E1 -9377.967,E2 -9377.967} C_VEL
LIN {X 0,Y 439.092,Z 558.048,A -85,B 0,C 180,E1 -9378.749,E2 -9378.749} C_VEL
LIN {X 0,Y 439.563,Z 543.962,A -85,B 0,C 180,E1 -9379.38,E2 -9379.38} C_VEL
LIN {X 0,Y 439.808,Z 529.162,A -85,B 0,C 180,E1 -9379.85,E2 -9379.85} C_VEL
LIN {X 0,Y 442.288,Z 457.46,A -85,B 0,C 180,E1 -9381.539,E2 -9381.539} C_VEL
LIN {X 0,Y 444.446,Z 408.583,A -85,B 0,C 180,E1 -9382.751,E2 -9382.751} C_VEL
LIN {X 0,Y 438.31,Z 397.125,A -85,B 0,C 180,E1 -9383.657,E2 -9383.657} C_VEL
LIN {X 0,Y 437.718,Z 394.994,A -85,B 0,C 180,E1 -9384.168,E2 -9384.168} C_VEL
LIN {X 0,Y 435.793,Z 387.816,A -85,B 0,C 180,E1 -9386.327,E2 -9386.327} C_VEL
LIN {X 0,Y 433.405,Z 380.32,A -85,B 0,C 180,E1 -9388.876,E2 -9388.876} C_VEL
LIN {X 0,Y 432.343,Z 377.301,A -85,B 0,C 180,E1 -9390.125,E2 -9390.125} C_VEL
LIN {X 0,Y 432.344,Z 377.257,A -85,B 0,C 180,E1 -9393.552,E2 -9393.552} C_VEL
LIN {X 0,Y 432.342,Z 377.258,A -85,B 0,C 180,E1 -9395.817,E2 -9395.817} C_VEL
LIN {X 0,Y 432.326,Z 377.258,A -85,B 0,C 180,E1 -9399.345,E2 -9399.345} C_VEL
LIN {X 0,Y 432.328,Z 377.26,A -85,B 0,C 180,E1 -9401.798,E2 -9401.798} C_VEL
LIN {X 0,Y 432.338,Z 377.258,A -85,B 0,C 180,E1 -9404.347,E2 -9404.347} C_VEL
LIN {X 0,Y 432.307,Z 377.262,A -85,B 0,C 180,E1 -9407.017,E2 -9407.017} C_VEL
LIN {X 0,Y 432.336,Z 377.446,A -85,B 0,C 180,E1 -9410.431,E2 -9410.431} C_VEL
LIN {X 0,Y 434.895,Z 384.101,A -85,B 0,C 180,E1 -9412.359,E2 -9412.359} C_VEL
LIN {X 0,Y 437.939,Z 392.438,A -85,B 0,C 180,E1 -9414.336,E2 -9414.336} C_VEL
LIN {X 0,Y 440.771,Z 401.923,A -85,B 0,C 180,E1 -9416.232,E2 -9416.232} C_VEL
LIN {X 0,Y 442.757,Z 410.446,A -85,B 0,C 180,E1 -9417.712,E2 -9417.712} C_VEL
LIN {X 0,Y 442.432,Z 415.414,A -85,B 0,C 180,E1 -9418.384,E2 -9418.384} C_VEL
LIN {X 0,Y 439.765,Z 440.161,A -85,B 0,C 180,E1 -9421.518,E2 -9421.518} C_VEL
LIN {X 0,Y 438.384,Z 457.106,A -85,B 0,C 180,E1 -9423.549,E2 -9423.549} C_VEL
LIN {X 0,Y 440.876,Z 474.759,A -85,B 0,C 180,E1 -9424.205,E2 -9424.205} C_VEL
LIN {X 0,Y 442.941,Z 496.412,A -85,B 0,C 180,E1 -9424.882,E2 -9424.882} C_VEL
LIN {X 0,Y 441.057,Z 620.619,A -85,B 0,C 180,E1 -9426.958,E2 -9426.958} C_VEL
LIN {X 0,Y 440.62,Z 643.144,A -85,B 0,C 180,E1 -9427.367,E2 -9427.367} C_VEL
LIN {X 0,Y 440.1,Z 657.552,A -85,B 0,C 180,E1 -9427.797,E2 -9427.797} C_VEL
LIN {X 0,Y 439.459,Z 670.527,A -85,B 0,C 180,E1 -9428.337,E2 -9428.337} C_VEL
LIN {X 0,Y 438.531,Z 684.775,A -85,B 0,C 180,E1 -9429.108,E2 -9429.108} C_VEL
LIN {X 0,Y 437.54,Z 698.325,A -85,B 0,C 180,E1 -9430.041,E2 -9430.041} C_VEL
LIN {X 0,Y 436.399,Z 712.051,A -85,B 0,C 180,E1 -9431.209,E2 -9431.209} C_VEL
LIN {X 0,Y 435.296,Z 724.887,A -85,B 0,C 180,E1 -9432.55,E2 -9432.55} C_VEL
LIN {X 0,Y 434.246,Z 736.548,A -85,B 0,C 180,E1 -9434.029,E2 -9434.029} C_VEL
LIN {X 0,Y 433.324,Z 747.281,A -85,B 0,C 180,E1 -9435.679,E2 -9435.679} C_VEL
LIN {X 0,Y 432.6,Z 755.911,A -85,B 0,C 180,E1 -9437.269,E2 -9437.269} C_VEL
LIN {X 0,Y 432.228,Z 762.591,A -85,B 0,C 180,E1 -9438.747,E2 -9438.747} C_VEL
LIN {X 0,Y 431.716,Z 769.651,A -85,B 0,C 180,E1 -9440.63,E2 -9440.63} C_VEL
LIN {X 0,Y 431.447,Z 775.195,A -85,B 0,C 180,E1 -9442.511,E2 -9442.511} C_VEL
LIN {X 0,Y 431.336,Z 779.383,A -85,B 0,C 180,E1 -9444.388,E2 -9444.388} C_VEL
LIN {X 0,Y 431.232,Z 782.316,A -85,B 0,C 180,E1 -9446.261,E2 -9446.261} C_VEL
LIN {X 0,Y 431.255,Z 784.063,A -85,B 0,C 180,E1 -9448.131,E2 -9448.131} C_VEL
LIN {X 0,Y 431.212,Z 784.658,A -85,B 0,C 180,E1 -9449.999,E2 -9449.999} C_VEL
LIN {X 0,Y 431.255,Z 784.061,A -85,B 0,C 180,E1 -9451.866,E2 -9451.866} C_VEL
LIN {X 0,Y 431.247,Z 782.312,A -85,B 0,C 180,E1 -9453.736,E2 -9453.736} C_VEL
LIN {X 0,Y 431.315,Z 779.383,A -85,B 0,C 180,E1 -9455.609,E2 -9455.609} C_VEL
LIN {X 0,Y 431.442,Z 775.201,A -85,B 0,C 180,E1 -9457.486,E2 -9457.486} C_VEL
LIN {X 0,Y 431.697,Z 769.654,A -85,B 0,C 180,E1 -9459.368,E2 -9459.368} C_VEL
LIN {X 0,Y 432.205,Z 762.587,A -85,B 0,C 180,E1 -9461.251,E2 -9461.251} C_VEL
LIN {X 0,Y 432.637,Z 754.918,A -85,B 0,C 180,E1 -9462.923,E2 -9462.923} C_VEL
LIN {X 0,Y 433.431,Z 745.87,A -85,B 0,C 180,E1 -9464.555,E2 -9464.555} C_VEL
LIN {X 0,Y 434.22,Z 736.548,A -85,B 0,C 180,E1 -9465.969,E2 -9465.969} C_VEL
LIN {X 0,Y 435.253,Z 724.965,A -85,B 0,C 180,E1 -9467.44,E2 -9467.44} C_VEL
LIN {X 0,Y 436.364,Z 712.057,A -85,B 0,C 180,E1 -9468.789,E2 -9468.789} C_VEL
LIN {X 0,Y 437.381,Z 699.868,A -85,B 0,C 180,E1 -9469.841,E2 -9469.841} C_VEL
LIN {X 0,Y 438.353,Z 686.647,A -85,B 0,C 180,E1 -9470.775,E2 -9470.775} C_VEL
LIN {X 0,Y 439.28,Z 672.118,A -85,B 0,C 180,E1 -9471.589,E2 -9471.589} C_VEL
LIN {X 0,Y 440.131,Z 657.028,A -85,B 0,C 180,E1 -9472.219,E2 -9472.219} C_VEL
LIN {X 0,Y 440.591,Z 643.119,A -85,B 0,C 180,E1 -9472.631,E2 -9472.631} C_VEL
LIN {X 0,Y 441.077,Z 616.98,A -85,B 0,C 180,E1 -9473.1,E2 -9473.1} C_VEL
LIN {X 0,Y 442.841,Z 495.694,A -85,B 0,C 180,E1 -9475.107,E2 -9475.107} C_VEL
LIN {X 0,Y 438.649,Z 464.479,A -85,B 0,C 180,E1 -9475.943,E2 -9475.943} C_VEL
LIN {X 0,Y 438.21,Z 459.187,A -85,B 0,C 180,E1 -9476.199,E2 -9476.199} C_VEL
LIN {X 0,Y 440.335,Z 427.699,A -85,B 0,C 180,E1 -9479.777,E2 -9479.777} C_VEL
LIN {X 0,Y 441.615,Z 409.893,A -85,B 0,C 180,E1 -9481.833,E2 -9481.833} C_VEL
LIN {X 0,Y 438.351,Z 397.736,A -85,B 0,C 180,E1 -9483.519,E2 -9483.519} C_VEL
LIN {X 0,Y 432.829,Z 379.165,A -85,B 0,C 180,E1 -9486.22,E2 -9486.22} C_VEL
LIN {X 0,Y 432.342,Z 377.415,A -85,B 0,C 180,E1 -9486.536,E2 -9486.536} C_VEL
LIN {X 0,Y 432.289,Z 377.263,A -85,B 0,C 180,E1 -9489.347,E2 -9489.347} C_VEL
LIN {X 0,Y 432.297,Z 377.262,A -85,B 0,C 180,E1 -9491.799,E2 -9491.799} C_VEL
LIN {X 0,Y 432.32,Z 377.261,A -85,B 0,C 180,E1 -9494.346,E2 -9494.346} C_VEL
LIN {X 0,Y 432.287,Z 377.238,A -85,B 0,C 180,E1 -9497.017,E2 -9497.017} C_VEL
LIN {X 0,Y 432.275,Z 377.255,A -85,B 0,C 180,E1 -9499.827,E2 -9499.827} C_VEL
LIN {X 0,Y 432.282,Z 377.247,A -85,B 0,C 180,E1 -9503.02,E2 -9503.02} C_VEL
LIN {X 0,Y 432.318,Z 377.233,A -85,B 0,C 180,E1 -9506.001,E2 -9506.001} C_VEL
LIN {X 0,Y 432.332,Z 377.254,A -85,B 0,C 180,E1 -9509.489,E2 -9509.489} C_VEL
LIN {X 0,Y 432.313,Z 377.253,A -85,B 0,C 180,E1 -9511.872,E2 -9511.872} C_VEL
LIN {X 0,Y 432.339,Z 377.243,A -85,B 0,C 180,E1 -9515.545,E2 -9515.545} C_VEL
LIN {X 0,Y 432.333,Z 377.248,A -85,B 0,C 180,E1 -9519.045,E2 -9519.045} C_VEL
LIN {X 0,Y 432.332,Z 377.254,A -85,B 0,C 180,E1 -9522.009,E2 -9522.009} C_VEL
LIN {X 0,Y 432.332,Z 377.244,A -85,B 0,C 180,E1 -9524.924,E2 -9524.924} C_VEL
LIN {X 0,Y 432.442,Z 377.241,A -85,B 0,C 180,E1 -9527.803,E2 -9527.803} C_VEL
LIN {X 0,Y 432.43,Z 377.236,A -85,B 0,C 180,E1 -9531.589,E2 -9531.589} C_VEL
LIN {X 0,Y 432.529,Z 377.228,A -85,B 0,C 180,E1 -9534.405,E2 -9534.405} C_VEL
LIN {X 0,Y 432.583,Z 377.223,A -85,B 0,C 180,E1 -9538.138,E2 -9538.138} C_VEL
LIN {X 0,Y 432.539,Z 377.218,A -85,B 0,C 180,E1 -9540.931,E2 -9540.931} C_VEL
LIN {X 0,Y 432.546,Z 377.228,A -85,B 0,C 180,E1 -9542.794,E2 -9542.794} C_VEL
LIN {X 0,Y 432.568,Z 377.219,A -85,B 0,C 180,E1 -9545.594,E2 -9545.594} C_VEL
LIN {X 0,Y 432.445,Z 377.239,A -85,B 0,C 180,E1 -9548.411,E2 -9548.411} C_VEL
LIN {X 0,Y 432.442,Z 377.229,A -85,B 0,C 180,E1 -9552.197,E2 -9552.197} C_VEL
LIN {X 0,Y 432.414,Z 377.239,A -85,B 0,C 180,E1 -9556.04,E2 -9556.04} C_VEL
LIN {X 0,Y 432.372,Z 377.247,A -85,B 0,C 180,E1 -9559.486,E2 -9559.486} C_VEL
LIN {X 0,Y 432.295,Z 377.263,A -85,B 0,C 180,E1 -9562.966,E2 -9562.966} C_VEL
LIN {X 0,Y 432.291,Z 377.253,A -85,B 0,C 180,E1 -9566.037,E2 -9566.037} C_VEL
LIN {X 0,Y 432.307,Z 377.254,A -85,B 0,C 180,E1 -9569.19,E2 -9569.19} C_VEL
LIN {X 0,Y 432.302,Z 377.258,A -85,B 0,C 180,E1 -9572.445,E2 -9572.445} C_VEL
LIN {X 0,Y 432.322,Z 377.253,A -85,B 0,C 180,E1 -9575.819,E2 -9575.819} C_VEL
LIN {X 0,Y 432.288,Z 377.261,A -85,B 0,C 180,E1 -9579.35,E2 -9579.35} C_VEL
LIN {X 0,Y 432.291,Z 377.249,A -85,B 0,C 180,E1 -9581.802,E2 -9581.802} C_VEL
LIN {X 0,Y 432.32,Z 377.257,A -85,B 0,C 180,E1 -9584.349,E2 -9584.349} C_VEL
LIN {X 0,Y 432.29,Z 377.249,A -85,B 0,C 180,E1 -9587.02,E2 -9587.02} C_VEL
LIN {X 0,Y 432.279,Z 377.252,A -85,B 0,C 180,E1 -9589.83,E2 -9589.83} C_VEL
LIN {X 0,Y 432.335,Z 377.486,A -85,B 0,C 180,E1 -9592.16,E2 -9592.16} C_VEL
LIN {X 0,Y 437.723,Z 394.04,A -85,B 0,C 180,E1 -9594.692,E2 -9594.692} C_VEL
LIN {X 0,Y 442.277,Z 410.154,A -85,B 0,C 180,E1 -9597.011,E2 -9597.011} C_VEL
LIN {X 0,Y 442.57,Z 412.561,A -85,B 0,C 180,E1 -9597.324,E2 -9597.324} C_VEL
LIN {X 0,Y 440.822,Z 442.436,A -85,B 0,C 180,E1 -9600.777,E2 -9600.777} C_VEL
LIN {X 0,Y 439.49,Z 469.292,A -85,B 0,C 180,E1 -9603.757,E2 -9603.757} C_VEL
LIN {X 0,Y 439.44,Z 472.376,A -85,B 0,C 180,E1 -9604.038,E2 -9604.038} C_VEL
LIN {X 0,Y 443.586,Z 498.267,A -85,B 0,C 180,E1 -9604.758,E2 -9604.758} C_VEL
LIN {X 0,Y 441.423,Z 635.933,A -85,B 0,C 180,E1 -9607.041,E2 -9607.041} C_VEL
LIN {X 0,Y 440.643,Z 641.77,A -85,B 0,C 180,E1 -9607.121,E2 -9607.121} C_VEL
LIN {X 0,Y 437.658,Z 651.213,A -85,B 0,C 180,E1 -9607.223,E2 -9607.223} C_VEL
LIN {X 0,Y 434.576,Z 660.519,A -85,B 0,C 180,E1 -9607.402,E2 -9607.402} C_VEL
LIN {X 0,Y 433.645,Z 666.135,A -85,B 0,C 180,E1 -9607.604,E2 -9607.604} C_VEL
LIN {X 0,Y 432.694,Z 681.401,A -85,B 0,C 180,E1 -9608.379,E2 -9608.379} C_VEL
LIN {X 0,Y 431.6,Z 694.963,A -85,B 0,C 180,E1 -9609.259,E2 -9609.259} C_VEL
LIN {X 0,Y 430.444,Z 708.163,A -85,B 0,C 180,E1 -9610.323,E2 -9610.323} C_VEL
LIN {X 0,Y 429.323,Z 720.393,A -85,B 0,C 180,E1 -9611.523,E2 -9611.523} C_VEL
LIN {X 0,Y 428.248,Z 731.448,A -85,B 0,C 180,E1 -9612.82,E2 -9612.82} C_VEL
LIN {X 0,Y 427.196,Z 741.739,A -85,B 0,C 180,E1 -9614.251,E2 -9614.251} C_VEL
LIN {X 0,Y 426.224,Z 751.808,A -85,B 0,C 180,E1 -9615.925,E2 -9615.925} C_VEL
LIN {X 0,Y 425.527,Z 760.168,A -85,B 0,C 180,E1 -9617.603,E2 -9617.603} C_VEL
LIN {X 0,Y 425.047,Z 766.223,A -85,B 0,C 180,E1 -9619.04,E2 -9619.04} C_VEL
LIN {X 0,Y 424.558,Z 772.852,A -85,B 0,C 180,E1 -9620.954,E2 -9620.954} C_VEL
LIN {X 0,Y 424.309,Z 778.039,A -85,B 0,C 180,E1 -9622.866,E2 -9622.866} C_VEL
LIN {X 0,Y 424.157,Z 781.016,A -85,B 0,C 180,E1 -9624.296,E2 -9624.296} C_VEL
LIN {X 0,Y 424.061,Z 783.949,A -85,B 0,C 180,E1 -9626.2,E2 -9626.2} C_VEL
LIN {X 0,Y 424.119,Z 785.713,A -85,B 0,C 180,E1 -9628.102,E2 -9628.102} C_VEL
LIN {X 0,Y 424.04,Z 786.326,A -85,B 0,C 180,E1 -9630.001,E2 -9630.001} C_VEL
LIN {X 0,Y 424.12,Z 785.76,A -85,B 0,C 180,E1 -9631.901,E2 -9631.901} C_VEL
LIN {X 0,Y 424.061,Z 784.059,A -85,B 0,C 180,E1 -9633.802,E2 -9633.802} C_VEL
LIN {X 0,Y 424.172,Z 781.184,A -85,B 0,C 180,E1 -9635.707,E2 -9635.707} C_VEL
LIN {X 0,Y 424.344,Z 777.07,A -85,B 0,C 180,E1 -9637.615,E2 -9637.615} C_VEL
LIN {X 0,Y 424.651,Z 771.619,A -85,B 0,C 180,E1 -9639.528,E2 -9639.528} C_VEL
LIN {X 0,Y 425.22,Z 764.679,A -85,B 0,C 180,E1 -9641.441,E2 -9641.441} C_VEL
LIN {X 0,Y 425.753,Z 757.284,A -85,B 0,C 180,E1 -9643.112,E2 -9643.112} C_VEL
LIN {X 0,Y 426.581,Z 748.281,A -85,B 0,C 180,E1 -9644.797,E2 -9644.797} C_VEL
LIN {X 0,Y 427.618,Z 737.459,A -85,B 0,C 180,E1 -9646.471,E2 -9646.471} C_VEL
LIN {X 0,Y 428.724,Z 726.333,A -85,B 0,C 180,E1 -9647.903,E2 -9647.903} C_VEL
LIN {X 0,Y 429.884,Z 714.156,A -85,B 0,C 180,E1 -9649.21,E2 -9649.21} C_VEL
LIN {X 0,Y 431.104,Z 700.729,A -85,B 0,C 180,E1 -9650.395,E2 -9650.395} C_VEL
LIN {X 0,Y 432.211,Z 687.606,A -85,B 0,C 180,E1 -9651.337,E2 -9651.337} C_VEL
LIN {X 0,Y 433.217,Z 673.979,A -85,B 0,C 180,E1 -9652.118,E2 -9652.118} C_VEL
LIN {X 0,Y 434.021,Z 658.879,A -85,B 0,C 180,E1 -9652.783,E2 -9652.783} C_VEL
LIN {X 0,Y 434.664,Z 643.939,A -85,B 0,C 180,E1 -9653.243,E2 -9653.243} C_VEL
LIN {X 0,Y 435.175,Z 619.889,A -85,B 0,C 180,E1 -9653.687,E2 -9653.687} C_VEL
LIN {X 0,Y 437.16,Z 498.6,A -85,B 0,C 180,E1 -9655.727,E2 -9655.727} C_VEL
LIN {X 0,Y 432.834,Z 471.94,A -85,B 0,C 180,E1 -9656.5,E2 -9656.5} C_VEL
LIN {X 0,Y 433.805,Z 451.072,A -85,B 0,C 180,E1 -9658.782,E2 -9658.782} C_VEL
LIN {X 0,Y 435.541,Z 421.789,A -85,B 0,C 180,E1 -9662.176,E2 -9662.176} C_VEL
LIN {X 0,Y 436.029,Z 414.271,A -85,B 0,C 180,E1 -9663.055,E2 -9663.055} C_VEL
LIN {X 0,Y 432.865,Z 402.259,A -85,B 0,C 180,E1 -9664.787,E2 -9664.787} C_VEL
LIN {X 0,Y 427.915,Z 386.272,A -85,B 0,C 180,E1 -9667.198,E2 -9667.198} C_VEL
LIN {X 0,Y 425.301,Z 378.323,A -85,B 0,C 180,E1 -9668.471,E2 -9668.471} C_VEL
LIN {X 0,Y 425.246,Z 378.126,A -85,B 0,C 180,E1 -9671.951,E2 -9671.951} C_VEL
LIN {X 0,Y 425.269,Z 378.122,A -85,B 0,C 180,E1 -9675.287,E2 -9675.287} C_VEL
LIN {X 0,Y 425.249,Z 378.133,A -85,B 0,C 180,E1 -9678.618,E2 -9678.618} C_VEL
LIN {X 0,Y 425.273,Z 378.135,A -85,B 0,C 180,E1 -9682.305,E2 -9682.305} C_VEL
LIN {X 0,Y 425.287,Z 378.114,A -85,B 0,C 180,E1 -9685.815,E2 -9685.815} C_VEL
LIN {X 0,Y 425.291,Z 378.137,A -85,B 0,C 180,E1 -9689.24,E2 -9689.24} C_VEL
LIN {X 0,Y 425.299,Z 378.135,A -85,B 0,C 180,E1 -9691.365,E2 -9691.365} C_VEL
LIN {X 0,Y 425.256,Z 378.14,A -85,B 0,C 180,E1 -9694.552,E2 -9694.552} C_VEL
LIN {X 0,Y 425.341,Z 378.269,A -85,B 0,C 180,E1 -9695.991,E2 -9695.991} C_VEL
LIN {X 0,Y 426.906,Z 385.37,A -85,B 0,C 180,E1 -9697.448,E2 -9697.448} C_VEL
LIN {X 0,Y 433.407,Z 403.163,A -85,B 0,C 180,E1 -9698.179,E2 -9698.179} C_VEL
LIN {X 0,Y 431.263,Z 506.4,A -85,B 0,C 180,E1 -9700.236,E2 -9700.236} C_VEL
LIN {X 0,Y 430.942,Z 528.569,A -85,B 0,C 180,E1 -9700.716,E2 -9700.716} C_VEL
LIN {X 0,Y 430.646,Z 543.881,A -85,B 0,C 180,E1 -9701.248,E2 -9701.248} C_VEL
LIN {X 0,Y 430.228,Z 557.737,A -85,B 0,C 180,E1 -9701.918,E2 -9701.918} C_VEL
LIN {X 0,Y 429.626,Z 571.113,A -85,B 0,C 180,E1 -9702.753,E2 -9702.753} C_VEL
LIN {X 0,Y 429.09,Z 583.336,A -85,B 0,C 180,E1 -9703.711,E2 -9703.711} C_VEL
LIN {X 0,Y 428.402,Z 595.767,A -85,B 0,C 180,E1 -9704.904,E2 -9704.904} C_VEL
LIN {X 0,Y 427.791,Z 606.11,A -85,B 0,C 180,E1 -9706.101,E2 -9706.101} C_VEL
LIN {X 0,Y 427.226,Z 615.588,A -85,B 0,C 180,E1 -9707.41,E2 -9707.41} C_VEL
LIN {X 0,Y 426.643,Z 624.256,A -85,B 0,C 180,E1 -9708.84,E2 -9708.84} C_VEL
LIN {X 0,Y 426.228,Z 632.551,A -85,B 0,C 180,E1 -9710.509,E2 -9710.509} C_VEL
LIN {X 0,Y 425.874,Z 638.448,A -85,B 0,C 180,E1 -9711.958,E2 -9711.958} C_VEL
LIN {X 0,Y 425.652,Z 643.161,A -85,B 0,C 180,E1 -9713.363,E2 -9713.363} C_VEL
LIN {X 0,Y 425.507,Z 646.969,A -85,B 0,C 180,E1 -9714.788,E2 -9714.788} C_VEL
LIN {X 0,Y 425.216,Z 649.933,A -85,B 0,C 180,E1 -9716.209,E2 -9716.209} C_VEL
LIN {X 0,Y 425.332,Z 651.419,A -85,B 0,C 180,E1 -9717.159,E2 -9717.159} C_VEL
LIN {X 0,Y 425.282,Z 653.386,A -85,B 0,C 180,E1 -9719.053,E2 -9719.053} C_VEL
LIN {X 0,Y 425.306,Z 653.976,A -85,B 0,C 180,E1 -9720.947,E2 -9720.947} C_VEL
LIN {X 0,Y 425.54,Z 653.151,A -85,B 0,C 180,E1 -9722.84,E2 -9722.84} C_VEL
LIN {X 0,Y 425.712,Z 650.915,A -85,B 0,C 180,E1 -9724.735,E2 -9724.735} C_VEL
LIN {X 0,Y 426.042,Z 648.244,A -85,B 0,C 180,E1 -9726.155,E2 -9726.155} C_VEL
LIN {X 0,Y 426.566,Z 643.363,A -85,B 0,C 180,E1 -9728.05,E2 -9728.05} C_VEL
LIN {X 0,Y 427.015,Z 638.545,A -85,B 0,C 180,E1 -9729.473,E2 -9729.473} C_VEL
LIN {X 0,Y 427.636,Z 631.583,A -85,B 0,C 180,E1 -9731.134,E2 -9731.134} C_VEL
LIN {X 0,Y 428.428,Z 622.819,A -85,B 0,C 180,E1 -9732.794,E2 -9732.794} C_VEL
LIN {X 0,Y 429.206,Z 613.57,A -85,B 0,C 180,E1 -9734.218,E2 -9734.218} C_VEL
LIN {X 0,Y 430.216,Z 602.332,A -85,B 0,C 180,E1 -9735.637,E2 -9735.637} C_VEL
LIN {X 0,Y 430.965,Z 590.894,A -85,B 0,C 180,E1 -9736.826,E2 -9736.826} C_VEL
LIN {X 0,Y 431.685,Z 578.203,A -85,B 0,C 180,E1 -9737.896,E2 -9737.896} C_VEL
LIN {X 0,Y 432.423,Z 564.785,A -85,B 0,C 180,E1 -9738.784,E2 -9738.784} C_VEL
LIN {X 0,Y 432.956,Z 551.166,A -85,B 0,C 180,E1 -9739.492,E2 -9739.492} C_VEL
LIN {X 0,Y 433.318,Z 536.176,A -85,B 0,C 180,E1 -9740.068,E2 -9740.068} C_VEL
LIN {X 0,Y 434.748,Z 490.054,A -85,B 0,C 180,E1 -9741.205,E2 -9741.205} C_VEL
LIN {X 0,Y 438.507,Z 411.366,A -85,B 0,C 180,E1 -9743.184,E2 -9743.184} C_VEL
LIN {X 0,Y 432.811,Z 400.729,A -85,B 0,C 180,E1 -9744.063,E2 -9744.063} C_VEL
LIN {X 0,Y 431.417,Z 398.013,A -85,B 0,C 180,E1 -9744.343,E2 -9744.343} C_VEL
LIN {X 0,Y 429.314,Z 390.213,A -85,B 0,C 180,E1 -9746.755,E2 -9746.755} C_VEL
LIN {X 0,Y 427.071,Z 383.182,A -85,B 0,C 180,E1 -9749.285,E2 -9749.285} C_VEL
LIN {X 0,Y 425.308,Z 378.214,A -85,B 0,C 180,E1 -9751.436,E2 -9751.436} C_VEL
LIN {X 0,Y 425.316,Z 378.133,A -85,B 0,C 180,E1 -9754.287,E2 -9754.287} C_VEL
LIN {X 0,Y 425.281,Z 378.137,A -85,B 0,C 180,E1 -9757.694,E2 -9757.694} C_VEL
LIN {X 0,Y 425.281,Z 378.137,A -85,B 0,C 180,E1 -9760.519,E2 -9760.519} C_VEL
LIN {X 0,Y 425.265,Z 378.14,A -85,B 0,C 180,E1 -9763.955,E2 -9763.955} C_VEL
LIN {X 0,Y 425.251,Z 378.141,A -85,B 0,C 180,E1 -9766.65,E2 -9766.65} C_VEL
LIN {X 0,Y 425.282,Z 378.284,A -85,B 0,C 180,E1 -9769.095,E2 -9769.095} C_VEL
LIN {X 0,Y 427.254,Z 383.429,A -85,B 0,C 180,E1 -9770.875,E2 -9770.875} C_VEL
LIN {X 0,Y 429.215,Z 388.382,A -85,B 0,C 180,E1 -9772.296,E2 -9772.296} C_VEL
LIN {X 0,Y 431.888,Z 395.859,A -85,B 0,C 180,E1 -9774.138,E2 -9774.138} C_VEL
LIN {X 0,Y 434.658,Z 405.271,A -85,B 0,C 180,E1 -9776.065,E2 -9776.065} C_VEL
LIN {X 0,Y 436.464,Z 413.598,A -85,B 0,C 180,E1 -9777.545,E2 -9777.545} C_VEL
LIN {X 0,Y 434.125,Z 433.192,A -85,B 0,C 180,E1 -9780.144,E2 -9780.144} C_VEL
LIN {X 0,Y 431.958,Z 456.087,A -85,B 0,C 180,E1 -9782.987,E2 -9782.987} C_VEL
LIN {X 0,Y 434.611,Z 474.922,A -85,B 0,C 180,E1 -9783.721,E2 -9783.721} C_VEL
LIN {X 0,Y 436.707,Z 497.45,A -85,B 0,C 180,E1 -9784.459,E2 -9784.459} C_VEL
LIN {X 0,Y 436.183,Z 515.873,A -85,B 0,C 180,E1 -9784.835,E2 -9784.835} C_VEL
LIN {X 0,Y 434.15,Z 640.818,A -85,B 0,C 180,E1 -9786.948,E2 -9786.948} C_VEL
LIN {X 0,Y 433.611,Z 655.651,A -85,B 0,C 180,E1 -9787.372,E2 -9787.372} C_VEL
LIN {X 0,Y 432.862,Z 669.849,A -85,B 0,C 180,E1 -9787.954,E2 -9787.954} C_VEL
LIN {X 0,Y 432.031,Z 682.845,A -85,B 0,C 180,E1 -9788.654,E2 -9788.654} C_VEL
LIN {X 0,Y 430.976,Z 696.789,A -85,B 0,C 180,E1 -9789.599,E2 -9789.599} C_VEL
LIN {X 0,Y 429.866,Z 709.513,A -85,B 0,C 180,E1 -9790.665,E2 -9790.665} C_VEL
LIN {X 0,Y 428.689,Z 722.253,A -85,B 0,C 180,E1 -9791.964,E2 -9791.964} C_VEL
LIN {X 0,Y 427.693,Z 733.046,A -85,B 0,C 180,E1 -9793.286,E2 -9793.286} C_VEL
LIN {X 0,Y 426.809,Z 742.93,A -85,B 0,C 180,E1 -9794.723,E2 -9794.723} C_VEL
LIN {X 0,Y 425.903,Z 752.577,A -85,B 0,C 180,E1 -9796.399,E2 -9796.399} C_VEL
LIN {X 0,Y 425.344,Z 760.6,A -85,B 0,C 180,E1 -9798.079,E2 -9798.079} C_VEL
LIN {X 0,Y 424.744,Z 768.062,A -85,B 0,C 180,E1 -9799.993,E2 -9799.993} C_VEL
LIN {X 0,Y 424.46,Z 773.974,A -85,B 0,C 180,E1 -9801.908,E2 -9801.908} C_VEL
LIN {X 0,Y 424.342,Z 777.995,A -85,B 0,C 180,E1 -9803.579,E2 -9803.579} C_VEL
LIN {X 0,Y 424.224,Z 781.016,A -85,B 0,C 180,E1 -9805.247,E2 -9805.247} C_VEL
LIN {X 0,Y 424.206,Z 783.349,A -85,B 0,C 180,E1 -9807.15,E2 -9807.15} C_VEL
LIN {X 0,Y 424.129,Z 784.52,A -85,B 0,C 180,E1 -9809.049,E2 -9809.049} C_VEL
LIN {X 0,Y 424.128,Z 784.519,A -85,B 0,C 180,E1 -9810.948,E2 -9810.948} C_VEL
LIN {X 0,Y 424.211,Z 783.345,A -85,B 0,C 180,E1 -9812.847,E2 -9812.847} C_VEL
LIN {X 0,Y 424.209,Z 781.013,A -85,B 0,C 180,E1 -9814.75,E2 -9814.75} C_VEL
LIN {X 0,Y 424.295,Z 777.469,A -85,B 0,C 180,E1 -9816.657,E2 -9816.657} C_VEL
LIN {X 0,Y 424.498,Z 772.622,A -85,B 0,C 180,E1 -9818.568,E2 -9818.568} C_VEL
LIN {X 0,Y 424.831,Z 766.337,A -85,B 0,C 180,E1 -9820.483,E2 -9820.483} C_VEL
LIN {X 0,Y 425.375,Z 759.548,A -85,B 0,C 180,E1 -9822.159,E2 -9822.159} C_VEL
LIN {X 0,Y 426.001,Z 751.339,A -85,B 0,C 180,E1 -9823.839,E2 -9823.839} C_VEL
LIN {X 0,Y 426.914,Z 741.43,A -85,B 0,C 180,E1 -9825.515,E2 -9825.515} C_VEL
LIN {X 0,Y 427.854,Z 731.267,A -85,B 0,C 180,E1 -9826.95,E2 -9826.95} C_VEL
LIN {X 0,Y 428.994,Z 719.138,A -85,B 0,C 180,E1 -9828.381,E2 -9828.381} C_VEL
LIN {X 0,Y 430.067,Z 706.939,A -85,B 0,C 180,E1 -9829.571,E2 -9829.571} C_VEL
LIN {X 0,Y 431.181,Z 693.623,A -85,B 0,C 180,E1 -9830.637,E2 -9830.637} C_VEL
LIN {X 0,Y 432.292,Z 678.859,A -85,B 0,C 180,E1 -9831.58,E2 -9831.58} C_VEL
LIN {X 0,Y 433.182,Z 664.205,A -85,B 0,C 180,E1 -9832.298,E2 -9832.298} C_VEL
LIN {X 0,Y 433.868,Z 648.562,A -85,B 0,C 180,E1 -9832.851,E2 -9832.851} C_VEL
LIN {X 0,Y 434.259,Z 633.221,A -85,B 0,C 180,E1 -9833.2,E2 -9833.2} C_VEL
LIN {X 0,Y 436.275,Z 506.468,A -85,B 0,C 180,E1 -9835.322,E2 -9835.322} C_VEL
LIN {X 0,Y 436.338,Z 495.82,A -85,B 0,C 180,E1 -9835.507,E2 -9835.507} C_VEL
LIN {X 0,Y 432.173,Z 464.592,A -85,B 0,C 180,E1 -9836.361,E2 -9836.361} C_VEL
LIN {X 0,Y 431.54,Z 457.451,A -85,B 0,C 180,E1 -9836.713,E2 -9836.713} C_VEL
LIN {X 0,Y 433.671,Z 427.606,A -85,B 0,C 180,E1 -9840.156,E2 -9840.156} C_VEL
LIN {X 0,Y 434.806,Z 411.126,A -85,B 0,C 180,E1 -9842.096,E2 -9842.096} C_VEL
LIN {X 0,Y 429.617,Z 392.823,A -85,B 0,C 180,E1 -9844.713,E2 -9844.713} C_VEL
LIN {X 0,Y 425.285,Z 378.371,A -85,B 0,C 180,E1 -9846.91,E2 -9846.91} C_VEL
LIN {X 0,Y 425.247,Z 378.141,A -85,B 0,C 180,E1 -9849.035,E2 -9849.035} C_VEL
LIN {X 0,Y 425.249,Z 378.141,A -85,B 0,C 180,E1 -9852.654,E2 -9852.654} C_VEL
LIN {X 0,Y 425.271,Z 378.134,A -85,B 0,C 180,E1 -9855.282,E2 -9855.282} C_VEL
LIN {X 0,Y 425.234,Z 378.116,A -85,B 0,C 180,E1 -9858.617,E2 -9858.617} C_VEL
LIN {X 0,Y 425.263,Z 378.136,A -85,B 0,C 180,E1 -9861.098,E2 -9861.098} C_VEL
LIN {X 0,Y 425.278,Z 378.099,A -85,B 0,C 180,E1 -9864.662,E2 -9864.662} C_VEL
LIN {X 0,Y 425.249,Z 378.137,A -85,B 0,C 180,E1 -9868.072,E2 -9868.072} C_VEL
LIN {X 0,Y 425.289,Z 378.126,A -85,B 0,C 180,E1 -9871.365,E2 -9871.365} C_VEL
LIN {X 0,Y 425.245,Z 378.131,A -85,B 0,C 180,E1 -9874.552,E2 -9874.552} C_VEL
LIN {X 0,Y 425.276,Z 378.134,A -85,B 0,C 180,E1 -9877.729,E2 -9877.729} C_VEL
LIN {X 0,Y 425.344,Z 378.119,A -85,B 0,C 180,E1 -9880.703,E2 -9880.703} C_VEL
LIN {X 0,Y 425.306,Z 378.128,A -85,B 0,C 180,E1 -9883.685,E2 -9883.685} C_VEL
LIN {X 0,Y 425.377,Z 378.122,A -85,B 0,C 180,E1 -9887.096,E2 -9887.096} C_VEL
LIN {X 0,Y 425.369,Z 378.112,A -85,B 0,C 180,E1 -9890.49,E2 -9890.49} C_VEL
LIN {X 0,Y 425.453,Z 378.11,A -85,B 0,C 180,E1 -9893.36,E2 -9893.36} C_VEL
LIN {X 0,Y 425.331,Z 378.114,A -85,B 0,C 180,E1 -9895.261,E2 -9895.261} C_VEL
LIN {X 0,Y 425.552,Z 378.099,A -85,B 0,C 180,E1 -9898.107,E2 -9898.107} C_VEL
LIN {X 0,Y 425.501,Z 378.094,A -85,B 0,C 180,E1 -9900.946,E2 -9900.946} C_VEL
LIN {X 0,Y 425.501,Z 378.106,A -85,B 0,C 180,E1 -9902.84,E2 -9902.84} C_VEL
LIN {X 0,Y 425.524,Z 378.097,A -85,B 0,C 180,E1 -9905.687,E2 -9905.687} C_VEL
LIN {X 0,Y 425.389,Z 378.12,A -85,B 0,C 180,E1 -9908.551,E2 -9908.551} C_VEL
LIN {X 0,Y 425.396,Z 378.108,A -85,B 0,C 180,E1 -9912.402,E2 -9912.402} C_VEL
LIN {X 0,Y 425.372,Z 378.113,A -85,B 0,C 180,E1 -9916.312,E2 -9916.312} C_VEL
LIN {X 0,Y 425.313,Z 378.126,A -85,B 0,C 180,E1 -9919.636,E2 -9919.636} C_VEL
LIN {X 0,Y 425.272,Z 378.13,A -85,B 0,C 180,E1 -9922.34,E2 -9922.34} C_VEL
LIN {X 0,Y 425.237,Z 378.131,A -85,B 0,C 180,E1 -9925.449,E2 -9925.449} C_VEL
LIN {X 0,Y 425.285,Z 378.129,A -85,B 0,C 180,E1 -9928.859,E2 -9928.859} C_VEL
LIN {X 0,Y 425.24,Z 378.139,A -85,B 0,C 180,E1 -9931.929,E2 -9931.929} C_VEL
LIN {X 0,Y 425.281,Z 378.132,A -85,B 0,C 180,E1 -9935.338,E2 -9935.338} C_VEL
LIN {X 0,Y 425.264,Z 378.125,A -85,B 0,C 180,E1 -9938.903,E2 -9938.903} C_VEL
LIN {X 0,Y 425.252,Z 378.123,A -85,B 0,C 180,E1 -9941.955,E2 -9941.955} C_VEL
LIN {X 0,Y 425.272,Z 378.135,A -85,B 0,C 180,E1 -9945.285,E2 -9945.285} C_VEL
LIN {X 0,Y 425.237,Z 378.145,A -85,B 0,C 180,E1 -9948.62,E2 -9948.62} C_VEL
LIN {X 0,Y 425.304,Z 378.312,A -85,B 0,C 180,E1 -9951.627,E2 -9951.627} C_VEL
LIN {X 0,Y 427.002,Z 383.534,A -85,B 0,C 180,E1 -9952.487,E2 -9952.487} C_VEL
LIN {X 0,Y 432.351,Z 400.182,A -85,B 0,C 180,E1 -9955.011,E2 -9955.011} C_VEL
LIN {X 0,Y 435.994,Z 413.573,A -85,B 0,C 180,E1 -9956.952,E2 -9956.952} C_VEL
LIN {X 0,Y 434.506,Z 438.797,A -85,B 0,C 180,E1 -9959.908,E2 -9959.908} C_VEL
LIN {X 0,Y 432.978,Z 468.225,A -85,B 0,C 180,E1 -9963.221,E2 -9963.221} C_VEL
LIN {X 0,Y 432.883,Z 472.268,A -85,B 0,C 180,E1 -9963.614,E2 -9963.614} C_VEL
LIN {X 0,Y 437.18,Z 498.914,A -85,B 0,C 180,E1 -9964.375,E2 -9964.375} C_VEL
LIN {X 0,Y 434.764,Z 640.065,A -85,B 0,C 180,E1 -9966.765,E2 -9966.765} C_VEL
LIN {X 0,Y 434.209,Z 655.878,A -85,B 0,C 180,E1 -9967.211,E2 -9967.211} C_VEL
LIN {X 0,Y 433.645,Z 666.135,A -85,B 0,C 180,E1 -9967.604,E2 -9967.604} C_VEL
LIN {X 0,Y 432.659,Z 671.801,A -85,B 0,C 180,E1 -9967.831,E2 -9967.831} C_VEL
LIN {X 0,Y 429.389,Z 680.962,A -85,B 0,C 180,E1 -9968.177,E2 -9968.177} C_VEL
LIN {X 0,Y 426.031,Z 689.672,A -85,B 0,C 180,E1 -9968.583,E2 -9968.583} C_VEL
LIN {X 0,Y 424.951,Z 694.776,A -85,B 0,C 180,E1 -9968.908,E2 -9968.908} C_VEL
LIN {X 0,Y 423.73,Z 708.139,A -85,B 0,C 180,E1 -9969.998,E2 -9969.998} C_VEL
LIN {X 0,Y 422.45,Z 721.369,A -85,B 0,C 180,E1 -9971.324,E2 -9971.324} C_VEL
LIN {X 0,Y 421.213,Z 733.293,A -85,B 0,C 180,E1 -9972.775,E2 -9972.775} C_VEL
LIN {X 0,Y 420.154,Z 743.321,A -85,B 0,C 180,E1 -9974.229,E2 -9974.229} C_VEL
LIN {X 0,Y 419.165,Z 753.12,A -85,B 0,C 180,E1 -9975.931,E2 -9975.931} C_VEL
LIN {X 0,Y 418.421,Z 762.298,A -85,B 0,C 180,E1 -9977.882,E2 -9977.882} C_VEL
LIN {X 0,Y 417.719,Z 769.713,A -85,B 0,C 180,E1 -9979.826,E2 -9979.826} C_VEL
LIN {X 0,Y 417.36,Z 775.603,A -85,B 0,C 180,E1 -9981.772,E2 -9981.772} C_VEL
LIN {X 0,Y 417.104,Z 780.249,A -85,B 0,C 180,E1 -9983.785,E2 -9983.785} C_VEL
LIN {X 0,Y 417.057,Z 782.619,A -85,B 0,C 180,E1 -9985.168,E2 -9985.168} C_VEL
LIN {X 0,Y 416.975,Z 784.96,A -85,B 0,C 180,E1 -9987.103,E2 -9987.103} C_VEL
LIN {X 0,Y 416.99,Z 786.154,A -85,B 0,C 180,E1 -9989.036,E2 -9989.036} C_VEL
LIN {X 0,Y 416.991,Z 786.17,A -85,B 0,C 180,E1 -9990.967,E2 -9990.967} C_VEL
LIN {X 0,Y 416.976,Z 785.038,A -85,B 0,C 180,E1 -9992.9,E2 -9992.9} C_VEL
LIN {X 0,Y 417.06,Z 782.757,A -85,B 0,C 180,E1 -9994.835,E2 -9994.835} C_VEL
LIN {X 0,Y 417.227,Z 779.271,A -85,B 0,C 180,E1 -9996.773,E2 -9996.773} C_VEL
LIN {X 0,Y 417.425,Z 774.503,A -85,B 0,C 180,E1 -9998.717,E2 -9998.717} C_VEL
LIN {X 0,Y 417.813,Z 768.329,A -85,B 0,C 180,E1 -10000.664,E2 -10000.664} C_VEL
LIN {X 0,Y 418.405,Z 761.662,A -85,B 0,C 180,E1 -10002.368,E2 -10002.368} C_VEL
LIN {X 0,Y 419.117,Z 753.578,A -85,B 0,C 180,E1 -10004.074,E2 -10004.074} C_VEL
LIN {X 0,Y 420.105,Z 743.873,A -85,B 0,C 180,E1 -10005.776,E2 -10005.776} C_VEL
LIN {X 0,Y 421.162,Z 733.93,A -85,B 0,C 180,E1 -10007.231,E2 -10007.231} C_VEL
LIN {X 0,Y 422.347,Z 722.123,A -85,B 0,C 180,E1 -10008.684,E2 -10008.684} C_VEL
LIN {X 0,Y 423.542,Z 710.339,A -85,B 0,C 180,E1 -10009.888,E2 -10009.888} C_VEL
LIN {X 0,Y 424.681,Z 697.614,A -85,B 0,C 180,E1 -10010.971,E2 -10010.971} C_VEL
LIN {X 0,Y 425.9,Z 683.717,A -85,B 0,C 180,E1 -10011.923,E2 -10011.923} C_VEL
LIN {X 0,Y 426.813,Z 669.818,A -85,B 0,C 180,E1 -10012.68,E2 -10012.68} C_VEL
LIN {X 0,Y 427.705,Z 654.709,A -85,B 0,C 180,E1 -10013.292,E2 -10013.292} C_VEL
LIN {X 0,Y 428.285,Z 639.805,A -85,B 0,C 180,E1 -10013.707,E2 -10013.707} C_VEL
LIN {X 0,Y 430.761,Z 500.703,A -85,B 0,C 180,E1 -10016.096,E2 -10016.096} C_VEL
LIN {X 0,Y 429.998,Z 494.267,A -85,B 0,C 180,E1 -10016.263,E2 -10016.263} C_VEL
LIN {X 0,Y 426.247,Z 471.948,A -85,B 0,C 180,E1 -10016.937,E2 -10016.937} C_VEL
LIN {X 0,Y 427.258,Z 451.991,A -85,B 0,C 180,E1 -10019.133,E2 -10019.133} C_VEL
LIN {X 0,Y 429.015,Z 423.644,A -85,B 0,C 180,E1 -10022.447,E2 -10022.447} C_VEL
LIN {X 0,Y 429.358,Z 415.629,A -85,B 0,C 180,E1 -10023.405,E2 -10023.405} C_VEL
LIN {X 0,Y 425.04,Z 400.229,A -85,B 0,C 180,E1 -10025.686,E2 -10025.686} C_VEL
LIN {X 0,Y 419.684,Z 383.469,A -85,B 0,C 180,E1 -10028.288,E2 -10028.288} C_VEL
LIN {X 0,Y 418.237,Z 379.197,A -85,B 0,C 180,E1 -10029.019,E2 -10029.019} C_VEL
LIN {X 0,Y 418.185,Z 379.005,A -85,B 0,C 180,E1 -10032.314,E2 -10032.314} C_VEL
LIN {X 0,Y 418.22,Z 379.001,A -85,B 0,C 180,E1 -10035.106,E2 -10035.106} C_VEL
LIN {X 0,Y 418.212,Z 379.016,A -85,B 0,C 180,E1 -10037.763,E2 -10037.763} C_VEL
LIN {X 0,Y 418.201,Z 378.998,A -85,B 0,C 180,E1 -10040.63,E2 -10040.63} C_VEL
LIN {X 0,Y 418.24,Z 379,A -85,B 0,C 180,E1 -10043.975,E2 -10043.975} C_VEL
LIN {X 0,Y 418.245,Z 379.005,A -85,B 0,C 180,E1 -10047.16,E2 -10047.16} C_VEL
LIN {X 0,Y 418.242,Z 379.013,A -85,B 0,C 180,E1 -10049.728,E2 -10049.728} C_VEL
LIN {X 0,Y 418.206,Z 379.018,A -85,B 0,C 180,E1 -10053.016,E2 -10053.016} C_VEL
LIN {X 0,Y 418.328,Z 379.227,A -85,B 0,C 180,E1 -10055.727,E2 -10055.727} C_VEL
LIN {X 0,Y 419.857,Z 386.119,A -85,B 0,C 180,E1 -10057.117,E2 -10057.117} C_VEL
LIN {X 0,Y 426.674,Z 404.384,A -85,B 0,C 180,E1 -10057.876,E2 -10057.876} C_VEL
LIN {X 0,Y 424.636,Z 500.374,A -85,B 0,C 180,E1 -10059.851,E2 -10059.851} C_VEL
LIN {X 0,Y 424.11,Z 528.552,A -85,B 0,C 180,E1 -10060.456,E2 -10060.456} C_VEL
LIN {X 0,Y 423.796,Z 544.196,A -85,B 0,C 180,E1 -10061.002,E2 -10061.002} C_VEL
LIN {X 0,Y 423.332,Z 559.192,A -85,B 0,C 180,E1 -10061.738,E2 -10061.738} C_VEL
LIN {X 0,Y 422.703,Z 572.409,A -85,B 0,C 180,E1 -10062.586,E2 -10062.586} C_VEL
LIN {X 0,Y 422.164,Z 584.562,A -85,B 0,C 180,E1 -10063.56,E2 -10063.56} C_VEL
LIN {X 0,Y 421.428,Z 596.954,A -85,B 0,C 180,E1 -10064.772,E2 -10064.772} C_VEL
LIN {X 0,Y 420.796,Z 607.955,A -85,B 0,C 180,E1 -10066.079,E2 -10066.079} C_VEL
LIN {X 0,Y 420.139,Z 617.518,A -85,B 0,C 180,E1 -10067.44,E2 -10067.44} C_VEL
LIN {X 0,Y 419.633,Z 626.046,A -85,B 0,C 180,E1 -10068.895,E2 -10068.895} C_VEL
LIN {X 0,Y 419.19,Z 634.237,A -85,B 0,C 180,E1 -10070.592,E2 -10070.592} C_VEL
LIN {X 0,Y 418.863,Z 640.813,A -85,B 0,C 180,E1 -10072.286,E2 -10072.286} C_VEL
LIN {X 0,Y 418.595,Z 645.308,A -85,B 0,C 180,E1 -10073.735,E2 -10073.735} C_VEL
LIN {X 0,Y 418.288,Z 648.934,A -85,B 0,C 180,E1 -10075.181,E2 -10075.181} C_VEL
LIN {X 0,Y 418.311,Z 652.375,A -85,B 0,C 180,E1 -10077.111,E2 -10077.111} C_VEL
LIN {X 0,Y 418.261,Z 654.415,A -85,B 0,C 180,E1 -10079.037,E2 -10079.037} C_VEL
LIN {X 0,Y 418.292,Z 655.065,A -85,B 0,C 180,E1 -10080.963,E2 -10080.963} C_VEL
LIN {X 0,Y 418.542,Z 654.299,A -85,B 0,C 180,E1 -10082.887,E2 -10082.887} C_VEL
LIN {X 0,Y 418.748,Z 652.142,A -85,B 0,C 180,E1 -10084.814,E2 -10084.814} C_VEL
LIN {X 0,Y 419.107,Z 649.513,A -85,B 0,C 180,E1 -10086.257,E2 -10086.257} C_VEL
LIN {X 0,Y 419.677,Z 644.692,A -85,B 0,C 180,E1 -10088.183,E2 -10088.183} C_VEL
LIN {X 0,Y 420.148,Z 639.906,A -85,B 0,C 180,E1 -10089.629,E2 -10089.629} C_VEL
LIN {X 0,Y 420.811,Z 632.978,A -85,B 0,C 180,E1 -10091.317,E2 -10091.317} C_VEL
LIN {X 0,Y 421.678,Z 624.328,A -85,B 0,C 180,E1 -10093.003,E2 -10093.003} C_VEL
LIN {X 0,Y 422.531,Z 615.204,A -85,B 0,C 180,E1 -10094.448,E2 -10094.448} C_VEL
LIN {X 0,Y 423.468,Z 605.458,A -85,B 0,C 180,E1 -10095.72,E2 -10095.72} C_VEL
LIN {X 0,Y 424.288,Z 593.905,A -85,B 0,C 180,E1 -10096.974,E2 -10096.974} C_VEL
LIN {X 0,Y 425.066,Z 581.71,A -85,B 0,C 180,E1 -10098.06,E2 -10098.06} C_VEL
LIN {X 0,Y 425.901,Z 568.21,A -85,B 0,C 180,E1 -10099.02,E2 -10099.02} C_VEL
LIN {X 0,Y 426.486,Z 554.3,A -85,B 0,C 180,E1 -10099.788,E2 -10099.788} C_VEL
LIN {X 0,Y 426.916,Z 538.867,A -85,B 0,C 180,E1 -10100.413,E2 -10100.413} C_VEL
LIN {X 0,Y 427.603,Z 513.04,A -85,B 0,C 180,E1 -10101.103,E2 -10101.103} C_VEL
LIN {X 0,Y 431.395,Z 434.717,A -85,B 0,C 180,E1 -10103.105,E2 -10103.105} C_VEL
LIN {X 0,Y 432.493,Z 413.591,A -85,B 0,C 180,E1 -10103.676,E2 -10103.676} C_VEL
LIN {X 0,Y 426.424,Z 402.512,A -85,B 0,C 180,E1 -10104.658,E2 -10104.658} C_VEL
LIN {X 0,Y 424.74,Z 399.518,A -85,B 0,C 180,E1 -10104.995,E2 -10104.995} C_VEL
LIN {X 0,Y 422.95,Z 392.796,A -85,B 0,C 180,E1 -10107.179,E2 -10107.179} C_VEL
LIN {X 0,Y 420.77,Z 386.143,A -85,B 0,C 180,E1 -10109.709,E2 -10109.709} C_VEL
LIN {X 0,Y 418.962,Z 381.395,A -85,B 0,C 180,E1 -10111.897,E2 -10111.897} C_VEL
LIN {X 0,Y 418.242,Z 379.064,A -85,B 0,C 180,E1 -10113.214,E2 -10113.214} C_VEL
LIN {X 0,Y 418.249,Z 379.013,A -85,B 0,C 180,E1 -10116.237,E2 -10116.237} C_VEL
LIN {X 0,Y 418.246,Z 379.014,A -85,B 0,C 180,E1 -10119.682,E2 -10119.682} C_VEL
LIN {X 0,Y 418.228,Z 379.015,A -85,B 0,C 180,E1 -10122.319,E2 -10122.319} C_VEL
LIN {X 0,Y 418.24,Z 379.014,A -85,B 0,C 180,E1 -10125.108,E2 -10125.108} C_VEL
LIN {X 0,Y 418.26,Z 379.242,A -85,B 0,C 180,E1 -10127.512,E2 -10127.512} C_VEL
LIN {X 0,Y 419.869,Z 383.309,A -85,B 0,C 180,E1 -10129.245,E2 -10129.245} C_VEL
LIN {X 0,Y 421.998,Z 388.58,A -85,B 0,C 180,E1 -10131.059,E2 -10131.059} C_VEL
LIN {X 0,Y 424.613,Z 395.598,A -85,B 0,C 180,E1 -10133.017,E2 -10133.017} C_VEL
LIN {X 0,Y 427.137,Z 403.446,A -85,B 0,C 180,E1 -10134.837,E2 -10134.837} C_VEL
LIN {X 0,Y 429.396,Z 412.272,A -85,B 0,C 180,E1 -10136.587,E2 -10136.587} C_VEL
LIN {X 0,Y 430.09,Z 416.683,A -85,B 0,C 180,E1 -10137.366,E2 -10137.366} C_VEL
LIN {X 0,Y 427.335,Z 437.508,A -85,B 0,C 180,E1 -10140.164,E2 -10140.164} C_VEL
LIN {X 0,Y 425.614,Z 454.921,A -85,B 0,C 180,E1 -10142.376,E2 -10142.376} C_VEL
LIN {X 0,Y 428.548,Z 475.845,A -85,B 0,C 180,E1 -10143.244,E2 -10143.244} C_VEL
LIN {X 0,Y 430.518,Z 498.354,A -85,B 0,C 180,E1 -10144.009,E2 -10144.009} C_VEL
LIN {X 0,Y 429.613,Z 524.172,A -85,B 0,C 180,E1 -10144.57,E2 -10144.57} C_VEL
LIN {X 0,Y 427.637,Z 640.945,A -85,B 0,C 180,E1 -10146.576,E2 -10146.576} C_VEL
LIN {X 0,Y 427.047,Z 656.117,A -85,B 0,C 180,E1 -10147.018,E2 -10147.018} C_VEL
LIN {X 0,Y 426.25,Z 671.107,A -85,B 0,C 180,E1 -10147.654,E2 -10147.654} C_VEL
LIN {X 0,Y 425.263,Z 684.863,A -85,B 0,C 180,E1 -10148.424,E2 -10148.424} C_VEL
LIN {X 0,Y 424.159,Z 698.397,A -85,B 0,C 180,E1 -10149.383,E2 -10149.383} C_VEL
LIN {X 0,Y 422.891,Z 712.112,A -85,B 0,C 180,E1 -10150.585,E2 -10150.585} C_VEL
LIN {X 0,Y 421.657,Z 724.904,A -85,B 0,C 180,E1 -10151.963,E2 -10151.963} C_VEL
LIN {X 0,Y 420.481,Z 736.595,A -85,B 0,C 180,E1 -10153.491,E2 -10153.491} C_VEL
LIN {X 0,Y 419.486,Z 747.323,A -85,B 0,C 180,E1 -10155.196,E2 -10155.196} C_VEL
LIN {X 0,Y 418.614,Z 755.975,A -85,B 0,C 180,E1 -10156.842,E2 -10156.842} C_VEL
LIN {X 0,Y 418.18,Z 762.627,A -85,B 0,C 180,E1 -10158.364,E2 -10158.364} C_VEL
LIN {X 0,Y 417.623,Z 769.685,A -85,B 0,C 180,E1 -10160.31,E2 -10160.31} C_VEL
LIN {X 0,Y 417.313,Z 775.227,A -85,B 0,C 180,E1 -10162.256,E2 -10162.256} C_VEL
LIN {X 0,Y 417.166,Z 779.413,A -85,B 0,C 180,E1 -10164.197,E2 -10164.197} C_VEL
LIN {X 0,Y 417.054,Z 782.345,A -85,B 0,C 180,E1 -10166.134,E2 -10166.134} C_VEL
LIN {X 0,Y 417.105,Z 784.091,A -85,B 0,C 180,E1 -10168.067,E2 -10168.067} C_VEL
LIN {X 0,Y 417.044,Z 784.686,A -85,B 0,C 180,E1 -10169.999,E2 -10169.999} C_VEL
LIN {X 0,Y 417.105,Z 784.089,A -85,B 0,C 180,E1 -10171.93,E2 -10171.93} C_VEL
LIN {X 0,Y 417.063,Z 782.34,A -85,B 0,C 180,E1 -10173.863,E2 -10173.863} C_VEL
LIN {X 0,Y 417.138,Z 779.411,A -85,B 0,C 180,E1 -10175.8,E2 -10175.8} C_VEL
LIN {X 0,Y 417.308,Z 775.23,A -85,B 0,C 180,E1 -10177.741,E2 -10177.741} C_VEL
LIN {X 0,Y 417.613,Z 769.683,A -85,B 0,C 180,E1 -10179.687,E2 -10179.687} C_VEL
LIN {X 0,Y 418.167,Z 762.618,A -85,B 0,C 180,E1 -10181.634,E2 -10181.634} C_VEL
LIN {X 0,Y 418.672,Z 755.424,A -85,B 0,C 180,E1 -10183.266,E2 -10183.266} C_VEL
LIN {X 0,Y 419.582,Z 745.905,A -85,B 0,C 180,E1 -10185.046,E2 -10185.046} C_VEL
LIN {X 0,Y 420.454,Z 736.586,A -85,B 0,C 180,E1 -10186.507,E2 -10186.507} C_VEL
LIN {X 0,Y 421.593,Z 725.112,A -85,B 0,C 180,E1 -10188.011,E2 -10188.011} C_VEL
LIN {X 0,Y 422.777,Z 713.338,A -85,B 0,C 180,E1 -10189.291,E2 -10189.291} C_VEL
LIN {X 0,Y 423.977,Z 699.923,A -85,B 0,C 180,E1 -10190.496,E2 -10190.496} C_VEL
LIN {X 0,Y 425.107,Z 686.711,A -85,B 0,C 180,E1 -10191.454,E2 -10191.454} C_VEL
LIN {X 0,Y 426.102,Z 672.197,A -85,B 0,C 180,E1 -10192.292,E2 -10192.292} C_VEL
LIN {X 0,Y 427.015,Z 656.864,A -85,B 0,C 180,E1 -10192.951,E2 -10192.951} C_VEL
LIN {X 0,Y 427.566,Z 642.152,A -85,B 0,C 180,E1 -10193.393,E2 -10193.393} C_VEL
LIN {X 0,Y 428.406,Z 595.696,A -85,B 0,C 180,E1 -10194.211,E2 -10194.211} C_VEL
LIN {X 0,Y 429.941,Z 496.781,A -85,B 0,C 180,E1 -10195.899,E2 -10195.899} C_VEL
LIN {X 0,Y 425.754,Z 465.368,A -85,B 0,C 180,E1 -10196.764,E2 -10196.764} C_VEL
LIN {X 0,Y 424.915,Z 455.515,A -85,B 0,C 180,E1 -10197.253,E2 -10197.253} C_VEL
LIN {X 0,Y 427.22,Z 425.131,A -85,B 0,C 180,E1 -10200.82,E2 -10200.82} C_VEL
LIN {X 0,Y 428.09,Z 413.215,A -85,B 0,C 180,E1 -10202.244,E2 -10202.244} C_VEL
LIN {X 0,Y 423.145,Z 395.652,A -85,B 0,C 180,E1 -10204.788,E2 -10204.788} C_VEL
LIN {X 0,Y 418.252,Z 379.193,A -85,B 0,C 180,E1 -10207.338,E2 -10207.338} C_VEL
LIN {X 0,Y 418.197,Z 379.019,A -85,B 0,C 180,E1 -10210.866,E2 -10210.866} C_VEL
LIN {X 0,Y 418.192,Z 379.018,A -85,B 0,C 180,E1 -10213.727,E2 -10213.727} C_VEL
LIN {X 0,Y 418.185,Z 379,A -85,B 0,C 180,E1 -10216.446,E2 -10216.446} C_VEL
LIN {X 0,Y 418.194,Z 379,A -85,B 0,C 180,E1 -10219.132,E2 -10219.132} C_VEL
LIN {X 0,Y 418.219,Z 379,A -85,B 0,C 180,E1 -10222.774,E2 -10222.774} C_VEL
LIN {X 0,Y 418.218,Z 378.991,A -85,B 0,C 180,E1 -10226.32,E2 -10226.32} C_VEL
LIN {X 0,Y 418.227,Z 379.012,A -85,B 0,C 180,E1 -10229.727,E2 -10229.727} C_VEL
LIN {X 0,Y 418.196,Z 379.016,A -85,B 0,C 180,E1 -10233.016,E2 -10233.016} C_VEL
LIN {X 0,Y 418.244,Z 379.003,A -85,B 0,C 180,E1 -10236.216,E2 -10236.216} C_VEL
LIN {X 0,Y 418.233,Z 379.003,A -85,B 0,C 180,E1 -10239.336,E2 -10239.336} C_VEL
LIN {X 0,Y 418.24,Z 379.014,A -85,B 0,C 180,E1 -10242.394,E2 -10242.394} C_VEL
LIN {X 0,Y 418.261,Z 378.996,A -85,B 0,C 180,E1 -10245.402,E2 -10245.402} C_VEL
LIN {X 0,Y 418.294,Z 379.006,A -85,B 0,C 180,E1 -10248.368,E2 -10248.368} C_VEL
LIN {X 0,Y 418.43,Z 378.984,A -85,B 0,C 180,E1 -10252.278,E2 -10252.278} C_VEL
LIN {X 0,Y 418.448,Z 378.984,A -85,B 0,C 180,E1 -10254.216,E2 -10254.216} C_VEL
LIN {X 0,Y 418.521,Z 378.974,A -85,B 0,C 180,E1 -10258.075,E2 -10258.075} C_VEL
LIN {X 0,Y 418.463,Z 378.97,A -85,B 0,C 180,E1 -10260.962,E2 -10260.962} C_VEL
LIN {X 0,Y 418.458,Z 378.984,A -85,B 0,C 180,E1 -10262.888,E2 -10262.888} C_VEL
LIN {X 0,Y 418.482,Z 378.974,A -85,B 0,C 180,E1 -10265.783,E2 -10265.783} C_VEL
LIN {X 0,Y 418.359,Z 378.997,A -85,B 0,C 180,E1 -10268.696,E2 -10268.696} C_VEL
LIN {X 0,Y 418.295,Z 378.989,A -85,B 0,C 180,E1 -10271.632,E2 -10271.632} C_VEL
LIN {X 0,Y 418.285,Z 379.007,A -85,B 0,C 180,E1 -10274.598,E2 -10274.598} C_VEL
LIN {X 0,Y 418.264,Z 379.001,A -85,B 0,C 180,E1 -10277.605,E2 -10277.605} C_VEL
LIN {X 0,Y 418.235,Z 379.004,A -85,B 0,C 180,E1 -10280.664,E2 -10280.664} C_VEL
LIN {X 0,Y 418.24,Z 379.01,A -85,B 0,C 180,E1 -10283.784,E2 -10283.784} C_VEL
LIN {X 0,Y 418.187,Z 379.021,A -85,B 0,C 180,E1 -10287.042,E2 -10287.042} C_VEL
LIN {X 0,Y 418.223,Z 379.011,A -85,B 0,C 180,E1 -10290.274,E2 -10290.274} C_VEL
LIN {X 0,Y 418.219,Z 379.014,A -85,B 0,C 180,E1 -10293.68,E2 -10293.68} C_VEL
LIN {X 0,Y 418.222,Z 378.988,A -85,B 0,C 180,E1 -10297.226,E2 -10297.226} C_VEL
LIN {X 0,Y 418.195,Z 379.014,A -85,B 0,C 180,E1 -10300.868,E2 -10300.868} C_VEL
LIN {X 0,Y 418.189,Z 379.009,A -85,B 0,C 180,E1 -10303.729,E2 -10303.729} C_VEL
LIN {X 0,Y 418.186,Z 379.004,A -85,B 0,C 180,E1 -10306.448,E2 -10306.448} C_VEL
LIN {X 0,Y 418.197,Z 379.013,A -85,B 0,C 180,E1 -10309.135,E2 -10309.135} C_VEL
LIN {X 0,Y 418.277,Z 379.227,A -85,B 0,C 180,E1 -10311.1,E2 -10311.1} C_VEL
LIN {X 0,Y 424.063,Z 396.773,A -85,B 0,C 180,E1 -10313.894,E2 -10313.894} C_VEL
LIN {X 0,Y 428.305,Z 411.471,A -85,B 0,C 180,E1 -10316.091,E2 -10316.091} C_VEL
LIN {X 0,Y 429.466,Z 416.048,A -85,B 0,C 180,E1 -10316.751,E2 -10316.751} C_VEL
LIN {X 0,Y 427.639,Z 445.24,A -85,B 0,C 180,E1 -10320.191,E2 -10320.191} C_VEL
LIN {X 0,Y 426.268,Z 471.546,A -85,B 0,C 180,E1 -10323.139,E2 -10323.139} C_VEL
LIN {X 0,Y 430.722,Z 499.057,A -85,B 0,C 180,E1 -10323.967,E2 -10323.967} C_VEL
LIN {X 0,Y 428.266,Z 639.978,A -85,B 0,C 180,E1 -10326.392,E2 -10326.392} C_VEL
LIN {X 0,Y 427.654,Z 655.986,A -85,B 0,C 180,E1 -10326.848,E2 -10326.848} C_VEL
LIN {X 0,Y 426.823,Z 669.885,A -85,B 0,C 180,E1 -10327.419,E2 -10327.419} C_VEL
LIN {X 0,Y 425.842,Z 684.248,A -85,B 0,C 180,E1 -10328.204,E2 -10328.204} C_VEL
LIN {X 0,Y 424.951,Z 694.776,A -85,B 0,C 180,E1 -10328.908,E2 -10328.908} C_VEL
LIN {X 0,Y 423.864,Z 699.96,A -85,B 0,C 180,E1 -10329.261,E2 -10329.261} C_VEL
LIN {X 0,Y 420.388,Z 708.229,A -85,B 0,C 180,E1 -10329.835,E2 -10329.835} C_VEL
LIN {X 0,Y 416.877,Z 716.192,A -85,B 0,C 180,E1 -10330.484,E2 -10330.484} C_VEL
LIN {X 0,Y 415.743,Z 720.852,A -85,B 0,C 180,E1 -10330.954,E2 -10330.954} C_VEL
LIN {X 0,Y 414.398,Z 733.274,A -85,B 0,C 180,E1 -10332.482,E2 -10332.482} C_VEL
LIN {X 0,Y 413.262,Z 743.304,A -85,B 0,C 180,E1 -10333.959,E2 -10333.959} C_VEL
LIN {X 0,Y 412.205,Z 753.105,A -85,B 0,C 180,E1 -10335.689,E2 -10335.689} C_VEL
LIN {X 0,Y 411.457,Z 761.239,A -85,B 0,C 180,E1 -10337.423,E2 -10337.423} C_VEL
LIN {X 0,Y 410.812,Z 767.981,A -85,B 0,C 180,E1 -10339.155,E2 -10339.155} C_VEL
LIN {X 0,Y 410.384,Z 774.232,A -85,B 0,C 180,E1 -10341.135,E2 -10341.135} C_VEL
LIN {X 0,Y 410.074,Z 779.064,A -85,B 0,C 180,E1 -10343.111,E2 -10343.111} C_VEL
LIN {X 0,Y 409.967,Z 782.605,A -85,B 0,C 180,E1 -10345.085,E2 -10345.085} C_VEL
LIN {X 0,Y 409.873,Z 784.947,A -85,B 0,C 180,E1 -10347.053,E2 -10347.053} C_VEL
LIN {X 0,Y 409.916,Z 786.14,A -85,B 0,C 180,E1 -10349.019,E2 -10349.019} C_VEL
LIN {X 0,Y 409.917,Z 786.156,A -85,B 0,C 180,E1 -10350.984,E2 -10350.984} C_VEL
LIN {X 0,Y 409.874,Z 785.024,A -85,B 0,C 180,E1 -10352.95,E2 -10352.95} C_VEL
LIN {X 0,Y 409.971,Z 782.742,A -85,B 0,C 180,E1 -10354.919,E2 -10354.919} C_VEL
LIN {X 0,Y 410.159,Z 779.256,A -85,B 0,C 180,E1 -10356.89,E2 -10356.89} C_VEL
LIN {X 0,Y 410.38,Z 774.486,A -85,B 0,C 180,E1 -10358.868,E2 -10358.868} C_VEL
LIN {X 0,Y 410.799,Z 768.311,A -85,B 0,C 180,E1 -10360.849,E2 -10360.849} C_VEL
LIN {X 0,Y 411.392,Z 761.643,A -85,B 0,C 180,E1 -10362.582,E2 -10362.582} C_VEL
LIN {X 0,Y 412.185,Z 753.558,A -85,B 0,C 180,E1 -10364.315,E2 -10364.315} C_VEL
LIN {X 0,Y 413.213,Z 743.85,A -85,B 0,C 180,E1 -10366.046,E2 -10366.046} C_VEL
LIN {X 0,Y 414.345,Z 733.905,A -85,B 0,C 180,E1 -10367.523,E2 -10367.523} C_VEL
LIN {X 0,Y 415.567,Z 722.095,A -85,B 0,C 180,E1 -10369,E2 -10369} C_VEL
LIN {X 0,Y 416.852,Z 710.307,A -85,B 0,C 180,E1 -10370.221,E2 -10370.221} C_VEL
LIN {X 0,Y 418.032,Z 697.576,A -85,B 0,C 180,E1 -10371.32,E2 -10371.32} C_VEL
LIN {X 0,Y 419.312,Z 683.671,A -85,B 0,C 180,E1 -10372.286,E2 -10372.286} C_VEL
LIN {X 0,Y 420.255,Z 669.76,A -85,B 0,C 180,E1 -10373.054,E2 -10373.054} C_VEL
LIN {X 0,Y 421.124,Z 655.489,A -85,B 0,C 180,E1 -10373.645,E2 -10373.645} C_VEL
LIN {X 0,Y 421.807,Z 639.679,A -85,B 0,C 180,E1 -10374.094,E2 -10374.094} C_VEL
LIN {X 0,Y 424.389,Z 500.801,A -85,B 0,C 180,E1 -10376.514,E2 -10376.514} C_VEL
LIN {X 0,Y 419.739,Z 471.743,A -85,B 0,C 180,E1 -10377.395,E2 -10377.395} C_VEL
LIN {X 0,Y 421.095,Z 446.88,A -85,B 0,C 180,E1 -10380.185,E2 -10380.185} C_VEL
LIN {X 0,Y 422.958,Z 418.426,A -85,B 0,C 180,E1 -10383.568,E2 -10383.568} C_VEL
LIN {X 0,Y 418.597,Z 402.866,A -85,B 0,C 180,E1 -10385.896,E2 -10385.896} C_VEL
LIN {X 0,Y 413.88,Z 387.89,A -85,B 0,C 180,E1 -10388.263,E2 -10388.263} C_VEL
LIN {X 0,Y 411.194,Z 380.15,A -85,B 0,C 180,E1 -10389.563,E2 -10389.563} C_VEL
LIN {X 0,Y 411.157,Z 379.881,A -85,B 0,C 180,E1 -10391.809,E2 -10391.809} C_VEL
LIN {X 0,Y 411.161,Z 379.877,A -85,B 0,C 180,E1 -10395.507,E2 -10395.507} C_VEL
LIN {X 0,Y 411.148,Z 379.885,A -85,B 0,C 180,E1 -10398.776,E2 -10398.776} C_VEL
LIN {X 0,Y 411.182,Z 379.891,A -85,B 0,C 180,E1 -10402.025,E2 -10402.025} C_VEL
LIN {X 0,Y 411.204,Z 379.863,A -85,B 0,C 180,E1 -10405.124,E2 -10405.124} C_VEL
LIN {X 0,Y 411.158,Z 379.893,A -85,B 0,C 180,E1 -10408.002,E2 -10408.002} C_VEL
LIN {X 0,Y 411.174,Z 379.894,A -85,B 0,C 180,E1 -10411.407,E2 -10411.407} C_VEL
LIN {X 0,Y 411.242,Z 379.942,A -85,B 0,C 180,E1 -10415.356,E2 -10415.356} C_VEL
LIN {X 0,Y 412.695,Z 386.449,A -85,B 0,C 180,E1 -10416.737,E2 -10416.737} C_VEL
LIN {X 0,Y 415.032,Z 392.787,A -85,B 0,C 180,E1 -10417.042,E2 -10417.042} C_VEL
LIN {X 0,Y 419.936,Z 405.778,A -85,B 0,C 180,E1 -10417.583,E2 -10417.583} C_VEL
LIN {X 0,Y 417.93,Z 495.833,A -85,B 0,C 180,E1 -10419.481,E2 -10419.481} C_VEL
LIN {X 0,Y 417.297,Z 528.54,A -85,B 0,C 180,E1 -10420.188,E2 -10420.188} C_VEL
LIN {X 0,Y 416.998,Z 543.471,A -85,B 0,C 180,E1 -10420.704,E2 -10420.704} C_VEL
LIN {X 0,Y 416.538,Z 558.398,A -85,B 0,C 180,E1 -10421.43,E2 -10421.43} C_VEL
LIN {X 0,Y 415.879,Z 572.01,A -85,B 0,C 180,E1 -10422.291,E2 -10422.291} C_VEL
LIN {X 0,Y 415.324,Z 584.44,A -85,B 0,C 180,E1 -10423.281,E2 -10423.281} C_VEL
LIN {X 0,Y 414.546,Z 597.033,A -85,B 0,C 180,E1 -10424.513,E2 -10424.513} C_VEL
LIN {X 0,Y 413.872,Z 608.418,A -85,B 0,C 180,E1 -10425.872,E2 -10425.872} C_VEL
LIN {X 0,Y 413.205,Z 617.898,A -85,B 0,C 180,E1 -10427.226,E2 -10427.226} C_VEL
LIN {X 0,Y 412.661,Z 626.549,A -85,B 0,C 180,E1 -10428.705,E2 -10428.705} C_VEL
LIN {X 0,Y 412.211,Z 634.849,A -85,B 0,C 180,E1 -10430.431,E2 -10430.431} C_VEL
LIN {X 0,Y 411.862,Z 641.525,A -85,B 0,C 180,E1 -10432.154,E2 -10432.154} C_VEL
LIN {X 0,Y 411.603,Z 646.109,A -85,B 0,C 180,E1 -10433.628,E2 -10433.628} C_VEL
LIN {X 0,Y 411.275,Z 649.812,A -85,B 0,C 180,E1 -10435.098,E2 -10435.098} C_VEL
LIN {X 0,Y 411.164,Z 651.773,A -85,B 0,C 180,E1 -10436.079,E2 -10436.079} C_VEL
LIN {X 0,Y 411.29,Z 653.335,A -85,B 0,C 180,E1 -10437.061,E2 -10437.061} C_VEL
LIN {X 0,Y 411.239,Z 655.441,A -85,B 0,C 180,E1 -10439.021,E2 -10439.021} C_VEL
LIN {X 0,Y 411.279,Z 656.161,A -85,B 0,C 180,E1 -10440.979,E2 -10440.979} C_VEL
LIN {X 0,Y 411.548,Z 655.469,A -85,B 0,C 180,E1 -10442.937,E2 -10442.937} C_VEL
LIN {X 0,Y 411.782,Z 653.385,A -85,B 0,C 180,E1 -10444.895,E2 -10444.895} C_VEL
LIN {X 0,Y 412.169,Z 650.791,A -85,B 0,C 180,E1 -10446.363,E2 -10446.363} C_VEL
LIN {X 0,Y 412.584,Z 647.355,A -85,B 0,C 180,E1 -10447.832,E2 -10447.832} C_VEL
LIN {X 0,Y 413.298,Z 641.298,A -85,B 0,C 180,E1 -10449.79,E2 -10449.79} C_VEL
LIN {X 0,Y 414.013,Z 634.472,A -85,B 0,C 180,E1 -10451.505,E2 -10451.505} C_VEL
LIN {X 0,Y 414.953,Z 625.907,A -85,B 0,C 180,E1 -10453.217,E2 -10453.217} C_VEL
LIN {X 0,Y 415.845,Z 616.842,A -85,B 0,C 180,E1 -10454.685,E2 -10454.685} C_VEL
LIN {X 0,Y 416.901,Z 606.402,A -85,B 0,C 180,E1 -10456.074,E2 -10456.074} C_VEL
LIN {X 0,Y 417.748,Z 595.862,A -85,B 0,C 180,E1 -10457.248,E2 -10457.248} C_VEL
LIN {X 0,Y 418.564,Z 583.859,A -85,B 0,C 180,E1 -10458.35,E2 -10458.35} C_VEL
LIN {X 0,Y 419.441,Z 570.572,A -85,B 0,C 180,E1 -10459.325,E2 -10459.325} C_VEL
LIN {X 0,Y 420.119,Z 556.169,A -85,B 0,C 180,E1 -10460.154,E2 -10460.154} C_VEL
LIN {X 0,Y 420.637,Z 540.764,A -85,B 0,C 180,E1 -10460.805,E2 -10460.805} C_VEL
LIN {X 0,Y 421.052,Z 524.169,A -85,B 0,C 180,E1 -10461.287,E2 -10461.287} C_VEL
LIN {X 0,Y 424.46,Z 454.159,A -85,B 0,C 180,E1 -10463.124,E2 -10463.124} C_VEL
LIN {X 0,Y 426.58,Z 416.102,A -85,B 0,C 180,E1 -10464.174,E2 -10464.174} C_VEL
LIN {X 0,Y 420.777,Z 405.665,A -85,B 0,C 180,E1 -10465.176,E2 -10465.176} C_VEL
LIN {X 0,Y 418.123,Z 401.01,A -85,B 0,C 180,E1 -10465.705,E2 -10465.705} C_VEL
LIN {X 0,Y 416.132,Z 393.843,A -85,B 0,C 180,E1 -10468.222,E2 -10468.222} C_VEL
LIN {X 0,Y 414.211,Z 388.21,A -85,B 0,C 180,E1 -10470.598,E2 -10470.598} C_VEL
LIN {X 0,Y 412.32,Z 382.942,A -85,B 0,C 180,E1 -10473.361,E2 -10473.361} C_VEL
LIN {X 0,Y 411.218,Z 379.973,A -85,B 0,C 180,E1 -10475.527,E2 -10475.527} C_VEL
LIN {X 0,Y 411.212,Z 379.889,A -85,B 0,C 180,E1 -10479.225,E2 -10479.225} C_VEL
LIN {X 0,Y 411.182,Z 379.894,A -85,B 0,C 180,E1 -10482.694,E2 -10482.694} C_VEL
LIN {X 0,Y 411.231,Z 380.04,A -85,B 0,C 180,E1 -10485.136,E2 -10485.136} C_VEL
LIN {X 0,Y 412.361,Z 383.039,A -85,B 0,C 180,E1 -10487.019,E2 -10487.019} C_VEL
LIN {X 0,Y 414.238,Z 387.343,A -85,B 0,C 180,E1 -10489.024,E2 -10489.024} C_VEL
LIN {X 0,Y 416.346,Z 392.784,A -85,B 0,C 180,E1 -10490.94,E2 -10490.94} C_VEL
LIN {X 0,Y 418.723,Z 399.352,A -85,B 0,C 180,E1 -10492.825,E2 -10492.825} C_VEL
LIN {X 0,Y 421.322,Z 407.677,A -85,B 0,C 180,E1 -10494.821,E2 -10494.821} C_VEL
LIN {X 0,Y 423.359,Z 416.347,A -85,B 0,C 180,E1 -10496.565,E2 -10496.565} C_VEL
LIN {X 0,Y 423.764,Z 419.386,A -85,B 0,C 180,E1 -10497.1,E2 -10497.1} C_VEL
LIN {X 0,Y 420.419,Z 443.225,A -85,B 0,C 180,E1 -10500.373,E2 -10500.373} C_VEL
LIN {X 0,Y 419.296,Z 453.635,A -85,B 0,C 180,E1 -10501.719,E2 -10501.719} C_VEL
LIN {X 0,Y 422.102,Z 472.466,A -85,B 0,C 180,E1 -10502.569,E2 -10502.569} C_VEL
LIN {X 0,Y 424.431,Z 498.173,A -85,B 0,C 180,E1 -10503.508,E2 -10503.508} C_VEL
LIN {X 0,Y 423.08,Z 533.083,A -85,B 0,C 180,E1 -10504.31,E2 -10504.31} C_VEL
LIN {X 0,Y 421.132,Z 641.071,A -85,B 0,C 180,E1 -10506.192,E2 -10506.192} C_VEL
LIN {X 0,Y 420.505,Z 656.62,A -85,B 0,C 180,E1 -10506.656,E2 -10506.656} C_VEL
LIN {X 0,Y 419.714,Z 670.356,A -85,B 0,C 180,E1 -10507.246,E2 -10507.246} C_VEL
LIN {X 0,Y 418.669,Z 684.907,A -85,B 0,C 180,E1 -10508.067,E2 -10508.067} C_VEL
LIN {X 0,Y 417.5,Z 698.433,A -85,B 0,C 180,E1 -10509.039,E2 -10509.039} C_VEL
LIN {X 0,Y 416.185,Z 712.142,A -85,B 0,C 180,E1 -10510.26,E2 -10510.26} C_VEL
LIN {X 0,Y 414.979,Z 723.705,A -85,B 0,C 180,E1 -10511.514,E2 -10511.514} C_VEL
LIN {X 0,Y 413.829,Z 734.868,A -85,B 0,C 180,E1 -10512.964,E2 -10512.964} C_VEL
LIN {X 0,Y 412.843,Z 744.452,A -85,B 0,C 180,E1 -10514.446,E2 -10514.446} C_VEL
LIN {X 0,Y 411.88,Z 753.843,A -85,B 0,C 180,E1 -10516.178,E2 -10516.178} C_VEL
LIN {X 0,Y 411.263,Z 761.641,A -85,B 0,C 180,E1 -10517.915,E2 -10517.915} C_VEL
LIN {X 0,Y 410.674,Z 768.096,A -85,B 0,C 180,E1 -10519.647,E2 -10519.647} C_VEL
LIN {X 0,Y 410.318,Z 774.005,A -85,B 0,C 180,E1 -10521.627,E2 -10521.627} C_VEL
LIN {X 0,Y 410.165,Z 778.562,A -85,B 0,C 180,E1 -10523.618,E2 -10523.618} C_VEL
LIN {X 0,Y 410.057,Z 781.046,A -85,B 0,C 180,E1 -10525.083,E2 -10525.083} C_VEL
LIN {X 0,Y 409.995,Z 783.377,A -85,B 0,C 180,E1 -10527.051,E2 -10527.051} C_VEL
LIN {X 0,Y 409.972,Z 784.547,A -85,B 0,C 180,E1 -10529.016,E2 -10529.016} C_VEL
LIN {X 0,Y 409.972,Z 784.547,A -85,B 0,C 180,E1 -10530.981,E2 -10530.981} C_VEL
LIN {X 0,Y 410.001,Z 783.372,A -85,B 0,C 180,E1 -10532.946,E2 -10532.946} C_VEL
LIN {X 0,Y 410.04,Z 781.04,A -85,B 0,C 180,E1 -10534.915,E2 -10534.915} C_VEL
LIN {X 0,Y 410.158,Z 777.497,A -85,B 0,C 180,E1 -10536.887,E2 -10536.887} C_VEL
LIN {X 0,Y 410.388,Z 772.65,A -85,B 0,C 180,E1 -10538.865,E2 -10538.865} C_VEL
LIN {X 0,Y 410.783,Z 766.367,A -85,B 0,C 180,E1 -10540.846,E2 -10540.846} C_VEL
LIN {X 0,Y 411.33,Z 759.58,A -85,B 0,C 180,E1 -10542.581,E2 -10542.581} C_VEL
LIN {X 0,Y 412.115,Z 751.372,A -85,B 0,C 180,E1 -10544.315,E2 -10544.315} C_VEL
LIN {X 0,Y 413.131,Z 741.466,A -85,B 0,C 180,E1 -10546.046,E2 -10546.046} C_VEL
LIN {X 0,Y 414.238,Z 731.306,A -85,B 0,C 180,E1 -10547.525,E2 -10547.525} C_VEL
LIN {X 0,Y 415.457,Z 719.181,A -85,B 0,C 180,E1 -10549.002,E2 -10549.002} C_VEL
LIN {X 0,Y 416.678,Z 706.988,A -85,B 0,C 180,E1 -10550.227,E2 -10550.227} C_VEL
LIN {X 0,Y 417.901,Z 693.68,A -85,B 0,C 180,E1 -10551.324,E2 -10551.324} C_VEL
LIN {X 0,Y 419.102,Z 678.931,A -85,B 0,C 180,E1 -10552.295,E2 -10552.295} C_VEL
LIN {X 0,Y 420.028,Z 665.027,A -85,B 0,C 180,E1 -10553,E2 -10553} C_VEL
LIN {X 0,Y 420.785,Z 649.676,A -85,B 0,C 180,E1 -10553.573,E2 -10553.573} C_VEL
LIN {X 0,Y 421.289,Z 633.458,A -85,B 0,C 180,E1 -10553.958,E2 -10553.958} C_VEL
LIN {X 0,Y 423.67,Z 498.876,A -85,B 0,C 180,E1 -10556.275,E2 -10556.275} C_VEL
LIN {X 0,Y 419.421,Z 466.601,A -85,B 0,C 180,E1 -10557.169,E2 -10557.169} C_VEL
LIN {X 0,Y 418.236,Z 453.514,A -85,B 0,C 180,E1 -10557.819,E2 -10557.819} C_VEL
LIN {X 0,Y 420.549,Z 425.182,A -85,B 0,C 180,E1 -10561.2,E2 -10561.2} C_VEL
LIN {X 0,Y 421.296,Z 416.413,A -85,B 0,C 180,E1 -10562.262,E2 -10562.262} C_VEL
LIN {X 0,Y 420.768,Z 412.855,A -85,B 0,C 180,E1 -10562.744,E2 -10562.744} C_VEL
LIN {X 0,Y 415.133,Z 393.339,A -85,B 0,C 180,E1 -10565.648,E2 -10565.648} C_VEL
LIN {X 0,Y 411.205,Z 380.054,A -85,B 0,C 180,E1 -10567.763,E2 -10567.763} C_VEL
LIN {X 0,Y 411.138,Z 379.897,A -85,B 0,C 180,E1 -10571.224,E2 -10571.224} C_VEL
LIN {X 0,Y 411.162,Z 379.897,A -85,B 0,C 180,E1 -10574.489,E2 -10574.489} C_VEL
LIN {X 0,Y 411.147,Z 379.864,A -85,B 0,C 180,E1 -10578.191,E2 -10578.191} C_VEL
LIN {X 0,Y 411.177,Z 379.892,A -85,B 0,C 180,E1 -10581.833,E2 -10581.833} C_VEL
LIN {X 0,Y 411.187,Z 379.852,A -85,B 0,C 180,E1 -10585.123,E2 -10585.123} C_VEL
LIN {X 0,Y 411.15,Z 379.892,A -85,B 0,C 180,E1 -10588.002,E2 -10588.002} C_VEL
LIN {X 0,Y 411.161,Z 379.885,A -85,B 0,C 180,E1 -10591.406,E2 -10591.406} C_VEL
LIN {X 0,Y 411.173,Z 379.879,A -85,B 0,C 180,E1 -10594.94,E2 -10594.94} C_VEL
LIN {X 0,Y 411.188,Z 379.89,A -85,B 0,C 180,E1 -10597.913,E2 -10597.913} C_VEL
LIN {X 0,Y 411.199,Z 379.885,A -85,B 0,C 180,E1 -10601.05,E2 -10601.05} C_VEL
LIN {X 0,Y 411.194,Z 379.883,A -85,B 0,C 180,E1 -10604.129,E2 -10604.129} C_VEL
LIN {X 0,Y 411.287,Z 379.877,A -85,B 0,C 180,E1 -10607.165,E2 -10607.165} C_VEL
LIN {X 0,Y 411.264,Z 379.868,A -85,B 0,C 180,E1 -10610.161,E2 -10610.161} C_VEL
LIN {X 0,Y 411.369,Z 379.866,A -85,B 0,C 180,E1 -10613.132,E2 -10613.132} C_VEL
LIN {X 0,Y 411.271,Z 379.865,A -85,B 0,C 180,E1 -10615.099,E2 -10615.099} C_VEL
LIN {X 0,Y 411.489,Z 379.85,A -85,B 0,C 180,E1 -10618.043,E2 -10618.043} C_VEL
LIN {X 0,Y 411.486,Z 379.84,A -85,B 0,C 180,E1 -10621.958,E2 -10621.958} C_VEL
LIN {X 0,Y 411.427,Z 379.852,A -85,B 0,C 180,E1 -10625.883,E2 -10625.883} C_VEL
LIN {X 0,Y 411.398,Z 379.855,A -85,B 0,C 180,E1 -10627.855,E2 -10627.855} C_VEL
LIN {X 0,Y 411.265,Z 379.864,A -85,B 0,C 180,E1 -10631.833,E2 -10631.833} C_VEL
LIN {X 0,Y 411.242,Z 379.88,A -85,B 0,C 180,E1 -10634.853,E2 -10634.853} C_VEL
LIN {X 0,Y 411.23,Z 379.878,A -85,B 0,C 180,E1 -10637.916,E2 -10637.916} C_VEL
LIN {X 0,Y 411.181,Z 379.88,A -85,B 0,C 180,E1 -10641.035,E2 -10641.035} C_VEL
LIN {X 0,Y 411.176,Z 379.892,A -85,B 0,C 180,E1 -10644.219,E2 -10644.219} C_VEL
LIN {X 0,Y 411.129,Z 379.897,A -85,B 0,C 180,E1 -10647.487,E2 -10647.487} C_VEL
LIN {X 0,Y 411.18,Z 379.886,A -85,B 0,C 180,E1 -10649.714,E2 -10649.714} C_VEL
LIN {X 0,Y 411.191,Z 379.888,A -85,B 0,C 180,E1 -10653.157,E2 -10653.157} C_VEL
LIN {X 0,Y 411.177,Z 379.87,A -85,B 0,C 180,E1 -10656.553,E2 -10656.553} C_VEL
LIN {X 0,Y 411.156,Z 379.894,A -85,B 0,C 180,E1 -10659.721,E2 -10659.721} C_VEL
LIN {X 0,Y 411.149,Z 379.877,A -85,B 0,C 180,E1 -10663.137,E2 -10663.137} C_VEL
LIN {X 0,Y 411.151,Z 379.885,A -85,B 0,C 180,E1 -10665.884,E2 -10665.884} C_VEL
LIN {X 0,Y 411.148,Z 379.886,A -85,B 0,C 180,E1 -10669.494,E2 -10669.494} C_VEL
LIN {X 0,Y 411.179,Z 380.103,A -85,B 0,C 180,E1 -10670.528,E2 -10670.528} C_VEL
LIN {X 0,Y 417.098,Z 397.603,A -85,B 0,C 180,E1 -10673.387,E2 -10673.387} C_VEL
LIN {X 0,Y 421.678,Z 413.493,A -85,B 0,C 180,E1 -10675.803,E2 -10675.803} C_VEL
LIN {X 0,Y 422.845,Z 417.868,A -85,B 0,C 180,E1 -10676.455,E2 -10676.455} C_VEL
LIN {X 0,Y 421.758,Z 435.351,A -85,B 0,C 180,E1 -10678.553,E2 -10678.553} C_VEL
LIN {X 0,Y 420.222,Z 461.059,A -85,B 0,C 180,E1 -10681.535,E2 -10681.535} C_VEL
LIN {X 0,Y 419.739,Z 471.757,A -85,B 0,C 180,E1 -10682.706,E2 -10682.706} C_VEL
LIN {X 0,Y 424.387,Z 500.976,A -85,B 0,C 180,E1 -10683.586,E2 -10683.586} C_VEL
LIN {X 0,Y 421.768,Z 639.892,A -85,B 0,C 180,E1 -10686.005,E2 -10686.005} C_VEL
LIN {X 0,Y 421.15,Z 655.549,A -85,B 0,C 180,E1 -10686.454,E2 -10686.454} C_VEL
LIN {X 0,Y 420.229,Z 670.55,A -85,B 0,C 180,E1 -10687.081,E2 -10687.081} C_VEL
LIN {X 0,Y 419.252,Z 684.217,A -85,B 0,C 180,E1 -10687.843,E2 -10687.843} C_VEL
LIN {X 0,Y 417.987,Z 698.008,A -85,B 0,C 180,E1 -10688.81,E2 -10688.81} C_VEL
LIN {X 0,Y 416.612,Z 711.932,A -85,B 0,C 180,E1 -10690.027,E2 -10690.027} C_VEL
LIN {X 0,Y 415.743,Z 720.852,A -85,B 0,C 180,E1 -10690.954,E2 -10690.954} C_VEL
LIN {X 0,Y 414.603,Z 725.435,A -85,B 0,C 180,E1 -10691.446,E2 -10691.446} C_VEL
LIN {X 0,Y 411.039,Z 732.725,A -85,B 0,C 180,E1 -10692.24,E2 -10692.24} C_VEL
LIN {X 0,Y 407.483,Z 739.581,A -85,B 0,C 180,E1 -10693.11,E2 -10693.11} C_VEL
LIN {X 0,Y 406.367,Z 743.482,A -85,B 0,C 180,E1 -10693.714,E2 -10693.714} C_VEL
LIN {X 0,Y 405.262,Z 753.089,A -85,B 0,C 180,E1 -10695.438,E2 -10695.438} C_VEL
LIN {X 0,Y 404.479,Z 761.224,A -85,B 0,C 180,E1 -10697.202,E2 -10697.202} C_VEL
LIN {X 0,Y 403.809,Z 767.967,A -85,B 0,C 180,E1 -10698.964,E2 -10698.964} C_VEL
LIN {X 0,Y 403.321,Z 774.218,A -85,B 0,C 180,E1 -10700.979,E2 -10700.979} C_VEL
LIN {X 0,Y 402.999,Z 779.05,A -85,B 0,C 180,E1 -10702.99,E2 -10702.99} C_VEL
LIN {X 0,Y 402.88,Z 782.592,A -85,B 0,C 180,E1 -10704.998,E2 -10704.998} C_VEL
LIN {X 0,Y 402.775,Z 784.933,A -85,B 0,C 180,E1 -10707.001,E2 -10707.001} C_VEL
LIN {X 0,Y 402.843,Z 786.127,A -85,B 0,C 180,E1 -10709.002,E2 -10709.002} C_VEL
LIN {X 0,Y 402.844,Z 786.142,A -85,B 0,C 180,E1 -10711.001,E2 -10711.001} C_VEL
LIN {X 0,Y 402.775,Z 785.009,A -85,B 0,C 180,E1 -10713.002,E2 -10713.002} C_VEL
LIN {X 0,Y 402.886,Z 782.727,A -85,B 0,C 180,E1 -10715.005,E2 -10715.005} C_VEL
LIN {X 0,Y 403.069,Z 779.24,A -85,B 0,C 180,E1 -10717.012,E2 -10717.012} C_VEL
LIN {X 0,Y 403.317,Z 774.47,A -85,B 0,C 180,E1 -10719.024,E2 -10719.024} C_VEL
LIN {X 0,Y 403.796,Z 768.293,A -85,B 0,C 180,E1 -10721.039,E2 -10721.039} C_VEL
LIN {X 0,Y 404.414,Z 761.624,A -85,B 0,C 180,E1 -10722.803,E2 -10722.803} C_VEL
LIN {X 0,Y 405.241,Z 753.537,A -85,B 0,C 180,E1 -10724.566,E2 -10724.566} C_VEL
LIN {X 0,Y 406.342,Z 743.828,A -85,B 0,C 180,E1 -10726.325,E2 -10726.325} C_VEL
LIN {X 0,Y 407.535,Z 733.881,A -85,B 0,C 180,E1 -10727.826,E2 -10727.826} C_VEL
LIN {X 0,Y 408.82,Z 722.067,A -85,B 0,C 180,E1 -10729.326,E2 -10729.326} C_VEL
LIN {X 0,Y 410.172,Z 710.275,A -85,B 0,C 180,E1 -10730.565,E2 -10730.565} C_VEL
LIN {X 0,Y 411.404,Z 697.538,A -85,B 0,C 180,E1 -10731.681,E2 -10731.681} C_VEL
LIN {X 0,Y 412.739,Z 683.626,A -85,B 0,C 180,E1 -10732.661,E2 -10732.661} C_VEL
LIN {X 0,Y 413.813,Z 668.607,A -85,B 0,C 180,E1 -10733.493,E2 -10733.493} C_VEL
LIN {X 0,Y 414.701,Z 654.55,A -85,B 0,C 180,E1 -10734.067,E2 -10734.067} C_VEL
LIN {X 0,Y 415.332,Z 639.554,A -85,B 0,C 180,E1 -10734.494,E2 -10734.494} C_VEL
LIN {X 0,Y 418.029,Z 501.785,A -85,B 0,C 180,E1 -10736.928,E2 -10736.928} C_VEL
LIN {X 0,Y 413.247,Z 471.705,A -85,B 0,C 180,E1 -10737.86,E2 -10737.86} C_VEL
LIN {X 0,Y 414.186,Z 453.729,A -85,B 0,C 180,E1 -10739.88,E2 -10739.88} C_VEL
LIN {X 0,Y 416.056,Z 426.22,A -85,B 0,C 180,E1 -10743.154,E2 -10743.154} C_VEL
LIN {X 0,Y 416.378,Z 420.474,A -85,B 0,C 180,E1 -10743.85,E2 -10743.85} C_VEL
LIN {X 0,Y 411.789,Z 404.02,A -85,B 0,C 180,E1 -10746.365,E2 -10746.365} C_VEL
LIN {X 0,Y 406.625,Z 388.026,A -85,B 0,C 180,E1 -10748.943,E2 -10748.943} C_VEL
LIN {X 0,Y 404.155,Z 380.964,A -85,B 0,C 180,E1 -10750.176,E2 -10750.176} C_VEL
LIN {X 0,Y 404.082,Z 380.768,A -85,B 0,C 180,E1 -10753.073,E2 -10753.073} C_VEL
LIN {X 0,Y 404.108,Z 380.756,A -85,B 0,C 180,E1 -10755.92,E2 -10755.92} C_VEL
LIN {X 0,Y 404.102,Z 380.764,A -85,B 0,C 180,E1 -10758.633,E2 -10758.633} C_VEL
LIN {X 0,Y 404.138,Z 380.761,A -85,B 0,C 180,E1 -10761.497,E2 -10761.497} C_VEL
LIN {X 0,Y 404.175,Z 380.738,A -85,B 0,C 180,E1 -10764.983,E2 -10764.983} C_VEL
LIN {X 0,Y 404.136,Z 380.769,A -85,B 0,C 180,E1 -10768.445,E2 -10768.445} C_VEL
LIN {X 0,Y 404.153,Z 380.767,A -85,B 0,C 180,E1 -10770.863,E2 -10770.863} C_VEL
LIN {X 0,Y 404.156,Z 380.769,A -85,B 0,C 180,E1 -10774.724,E2 -10774.724} C_VEL
LIN {X 0,Y 404.199,Z 380.992,A -85,B 0,C 180,E1 -10775.124,E2 -10775.124} C_VEL
LIN {X 0,Y 405.61,Z 387.097,A -85,B 0,C 180,E1 -10776.392,E2 -10776.392} C_VEL
LIN {X 0,Y 413.235,Z 407.373,A -85,B 0,C 180,E1 -10777.286,E2 -10777.286} C_VEL
LIN {X 0,Y 411.007,Z 503.049,A -85,B 0,C 180,E1 -10779.349,E2 -10779.349} C_VEL
LIN {X 0,Y 410.468,Z 530.628,A -85,B 0,C 180,E1 -10779.974,E2 -10779.974} C_VEL
LIN {X 0,Y 410.098,Z 546.21,A -85,B 0,C 180,E1 -10780.544,E2 -10780.544} C_VEL
LIN {X 0,Y 409.588,Z 560.975,A -85,B 0,C 180,E1 -10781.297,E2 -10781.297} C_VEL
LIN {X 0,Y 408.898,Z 574.988,A -85,B 0,C 180,E1 -10782.237,E2 -10782.237} C_VEL
LIN {X 0,Y 408.328,Z 587.018,A -85,B 0,C 180,E1 -10783.244,E2 -10783.244} C_VEL
LIN {X 0,Y 407.534,Z 599.338,A -85,B 0,C 180,E1 -10784.496,E2 -10784.496} C_VEL
LIN {X 0,Y 406.895,Z 610.193,A -85,B 0,C 180,E1 -10785.835,E2 -10785.835} C_VEL
LIN {X 0,Y 406.18,Z 619.831,A -85,B 0,C 180,E1 -10787.255,E2 -10787.255} C_VEL
LIN {X 0,Y 405.657,Z 628.339,A -85,B 0,C 180,E1 -10788.761,E2 -10788.761} C_VEL
LIN {X 0,Y 405.177,Z 636.522,A -85,B 0,C 180,E1 -10790.515,E2 -10790.515} C_VEL
LIN {X 0,Y 404.839,Z 642.207,A -85,B 0,C 180,E1 -10792.017,E2 -10792.017} C_VEL
LIN {X 0,Y 404.593,Z 646.88,A -85,B 0,C 180,E1 -10793.517,E2 -10793.517} C_VEL
LIN {X 0,Y 404.264,Z 650.667,A -85,B 0,C 180,E1 -10795.013,E2 -10795.013} C_VEL
LIN {X 0,Y 404.137,Z 652.67,A -85,B 0,C 180,E1 -10796.011,E2 -10796.011} C_VEL
LIN {X 0,Y 404.268,Z 654.274,A -85,B 0,C 180,E1 -10797.01,E2 -10797.01} C_VEL
LIN {X 0,Y 404.217,Z 656.463,A -85,B 0,C 180,E1 -10799.004,E2 -10799.004} C_VEL
LIN {X 0,Y 404.267,Z 657.265,A -85,B 0,C 180,E1 -10800.996,E2 -10800.996} C_VEL
LIN {X 0,Y 404.555,Z 656.64,A -85,B 0,C 180,E1 -10802.987,E2 -10802.987} C_VEL
LIN {X 0,Y 404.814,Z 654.62,A -85,B 0,C 180,E1 -10804.98,E2 -10804.98} C_VEL
LIN {X 0,Y 404.986,Z 653.069,A -85,B 0,C 180,E1 -10805.976,E2 -10805.976} C_VEL
LIN {X 0,Y 405.595,Z 649.938,A -85,B 0,C 180,E1 -10807.467,E2 -10807.467} C_VEL
LIN {X 0,Y 406.174,Z 644.947,A -85,B 0,C 180,E1 -10809.296,E2 -10809.296} C_VEL
LIN {X 0,Y 407.002,Z 638.095,A -85,B 0,C 180,E1 -10811.201,E2 -10811.201} C_VEL
LIN {X 0,Y 407.914,Z 630.08,A -85,B 0,C 180,E1 -10812.943,E2 -10812.943} C_VEL
LIN {X 0,Y 408.89,Z 621.718,A -85,B 0,C 180,E1 -10814.432,E2 -10814.432} C_VEL
LIN {X 0,Y 409.774,Z 613.418,A -85,B 0,C 180,E1 -10815.672,E2 -10815.672} C_VEL
LIN {X 0,Y 410.818,Z 602.436,A -85,B 0,C 180,E1 -10817.035,E2 -10817.035} C_VEL
LIN {X 0,Y 411.803,Z 590.236,A -85,B 0,C 180,E1 -10818.276,E2 -10818.276} C_VEL
LIN {X 0,Y 412.653,Z 578.372,A -85,B 0,C 180,E1 -10819.268,E2 -10819.268} C_VEL
LIN {X 0,Y 413.537,Z 564.23,A -85,B 0,C 180,E1 -10820.207,E2 -10820.207} C_VEL
LIN {X 0,Y 414.169,Z 551.065,A -85,B 0,C 180,E1 -10820.876,E2 -10820.876} C_VEL
LIN {X 0,Y 414.522,Z 535.763,A -85,B 0,C 180,E1 -10821.451,E2 -10821.451} C_VEL
LIN {X 0,Y 416.571,Z 489.81,A -85,B 0,C 180,E1 -10822.701,E2 -10822.701} C_VEL
LIN {X 0,Y 420.922,Z 419.145,A -85,B 0,C 180,E1 -10824.672,E2 -10824.672} C_VEL
LIN {X 0,Y 416.53,Z 411.008,A -85,B 0,C 180,E1 -10825.468,E2 -10825.468} C_VEL
LIN {X 0,Y 411.594,Z 402.736,A -85,B 0,C 180,E1 -10826.444,E2 -10826.444} C_VEL
LIN {X 0,Y 409.858,Z 396.643,A -85,B 0,C 180,E1 -10828.694,E2 -10828.694} C_VEL
LIN {X 0,Y 408.077,Z 391.289,A -85,B 0,C 180,E1 -10831.109,E2 -10831.109} C_VEL
LIN {X 0,Y 406.516,Z 386.921,A -85,B 0,C 180,E1 -10833.589,E2 -10833.589} C_VEL
LIN {X 0,Y 405.629,Z 384.42,A -85,B 0,C 180,E1 -10835.477,E2 -10835.477} C_VEL
LIN {X 0,Y 404.705,Z 382.797,A -85,B 0,C 180,E1 -10837.431,E2 -10837.431} C_VEL
LIN {X 0,Y 404.44,Z 382.079,A -85,B 0,C 180,E1 -10838.724,E2 -10838.724} C_VEL
LIN {X 0,Y 404.35,Z 381.765,A -85,B 0,C 180,E1 -10840.113,E2 -10840.113} C_VEL
LIN {X 0,Y 404.6,Z 382.508,A -85,B 0,C 180,E1 -10842.644,E2 -10842.644} C_VEL
LIN {X 0,Y 405.549,Z 384.222,A -85,B 0,C 180,E1 -10844.722,E2 -10844.722} C_VEL
LIN {X 0,Y 407.141,Z 388.03,A -85,B 0,C 180,E1 -10847.18,E2 -10847.18} C_VEL
LIN {X 0,Y 408.993,Z 392.548,A -85,B 0,C 180,E1 -10849.232,E2 -10849.232} C_VEL
LIN {X 0,Y 411.392,Z 398.81,A -85,B 0,C 180,E1 -10851.404,E2 -10851.404} C_VEL
LIN {X 0,Y 414.005,Z 406.632,A -85,B 0,C 180,E1 -10853.547,E2 -10853.547} C_VEL
LIN {X 0,Y 416.356,Z 415.365,A -85,B 0,C 180,E1 -10855.537,E2 -10855.537} C_VEL
LIN {X 0,Y 417.384,Z 420.386,A -85,B 0,C 180,E1 -10856.532,E2 -10856.532} C_VEL
LIN {X 0,Y 417.439,Z 422.067,A -85,B 0,C 180,E1 -10856.826,E2 -10856.826} C_VEL
LIN {X 0,Y 414.065,Z 444.319,A -85,B 0,C 180,E1 -10859.955,E2 -10859.955} C_VEL
LIN {X 0,Y 413.103,Z 452.468,A -85,B 0,C 180,E1 -10861.025,E2 -10861.025} C_VEL
LIN {X 0,Y 415.789,Z 470.406,A -85,B 0,C 180,E1 -10861.897,E2 -10861.897} C_VEL
LIN {X 0,Y 417.666,Z 488.9,A -85,B 0,C 180,E1 -10862.638,E2 -10862.638} C_VEL
LIN {X 0,Y 418.411,Z 499.833,A -85,B 0,C 180,E1 -10863.029,E2 -10863.029} C_VEL
LIN {X 0,Y 416.606,Z 542.314,A -85,B 0,C 180,E1 -10864.051,E2 -10864.051} C_VEL
LIN {X 0,Y 414.654,Z 641.195,A -85,B 0,C 180,E1 -10865.797,E2 -10865.797} C_VEL
LIN {X 0,Y 414.016,Z 656.446,A -85,B 0,C 180,E1 -10866.258,E2 -10866.258} C_VEL
LIN {X 0,Y 413.169,Z 670.464,A -85,B 0,C 180,E1 -10866.867,E2 -10866.867} C_VEL
LIN {X 0,Y 412.086,Z 684.95,A -85,B 0,C 180,E1 -10867.698,E2 -10867.698} C_VEL
LIN {X 0,Y 410.863,Z 698.469,A -85,B 0,C 180,E1 -10868.684,E2 -10868.684} C_VEL
LIN {X 0,Y 409.467,Z 712.172,A -85,B 0,C 180,E1 -10869.922,E2 -10869.922} C_VEL
LIN {X 0,Y 408.14,Z 724.41,A -85,B 0,C 180,E1 -10871.276,E2 -10871.276} C_VEL
LIN {X 0,Y 406.985,Z 734.892,A -85,B 0,C 180,E1 -10872.668,E2 -10872.668} C_VEL
LIN {X 0,Y 405.947,Z 744.473,A -85,B 0,C 180,E1 -10874.175,E2 -10874.175} C_VEL
LIN {X 0,Y 404.938,Z 753.862,A -85,B 0,C 180,E1 -10875.936,E2 -10875.936} C_VEL
LIN {X 0,Y 404.266,Z 761.659,A -85,B 0,C 180,E1 -10877.703,E2 -10877.703} C_VEL
LIN {X 0,Y 403.632,Z 768.113,A -85,B 0,C 180,E1 -10879.464,E2 -10879.464} C_VEL
LIN {X 0,Y 403.264,Z 774.021,A -85,B 0,C 180,E1 -10881.48,E2 -10881.48} C_VEL
LIN {X 0,Y 403.057,Z 778.86,A -85,B 0,C 180,E1 -10883.664,E2 -10883.664} C_VEL
LIN {X 0,Y 402.968,Z 781.061,A -85,B 0,C 180,E1 -10884.996,E2 -10884.996} C_VEL
LIN {X 0,Y 402.892,Z 783.391,A -85,B 0,C 180,E1 -10886.999,E2 -10886.999} C_VEL
LIN {X 0,Y 402.897,Z 784.561,A -85,B 0,C 180,E1 -10888.999,E2 -10888.999} C_VEL
LIN {X 0,Y 402.897,Z 784.56,A -85,B 0,C 180,E1 -10890.998,E2 -10890.998} C_VEL
LIN {X 0,Y 402.898,Z 783.386,A -85,B 0,C 180,E1 -10892.998,E2 -10892.998} C_VEL
LIN {X 0,Y 402.951,Z 781.054,A -85,B 0,C 180,E1 -10895.001,E2 -10895.001} C_VEL
LIN {X 0,Y 403.069,Z 777.511,A -85,B 0,C 180,E1 -10897.009,E2 -10897.009} C_VEL
LIN {X 0,Y 403.323,Z 772.665,A -85,B 0,C 180,E1 -10899.021,E2 -10899.021} C_VEL
LIN {X 0,Y 403.776,Z 766.382,A -85,B 0,C 180,E1 -10901.036,E2 -10901.036} C_VEL
LIN {X 0,Y 404.344,Z 759.595,A -85,B 0,C 180,E1 -10902.802,E2 -10902.802} C_VEL
LIN {X 0,Y 405.187,Z 751.389,A -85,B 0,C 180,E1 -10904.565,E2 -10904.565} C_VEL
LIN {X 0,Y 406.259,Z 741.484,A -85,B 0,C 180,E1 -10906.325,E2 -10906.325} C_VEL
LIN {X 0,Y 407.439,Z 731.325,A -85,B 0,C 180,E1 -10907.827,E2 -10907.827} C_VEL
LIN {X 0,Y 408.703,Z 719.203,A -85,B 0,C 180,E1 -10909.329,E2 -10909.329} C_VEL
LIN {X 0,Y 409.99,Z 707.013,A -85,B 0,C 180,E1 -10910.572,E2 -10910.572} C_VEL
LIN {X 0,Y 411.277,Z 693.709,A -85,B 0,C 180,E1 -10911.685,E2 -10911.685} C_VEL
LIN {X 0,Y 412.55,Z 678.966,A -85,B 0,C 180,E1 -10912.668,E2 -10912.668} C_VEL
LIN {X 0,Y 413.559,Z 664.464,A -85,B 0,C 180,E1 -10913.412,E2 -10913.412} C_VEL
LIN {X 0,Y 414.342,Z 648.937,A -85,B 0,C 180,E1 -10913.989,E2 -10913.989} C_VEL
LIN {X 0,Y 414.817,Z 633.574,A -85,B 0,C 180,E1 -10914.356,E2 -10914.356} C_VEL
LIN {X 0,Y 417.262,Z 500.412,A -85,B 0,C 180,E1 -10916.684,E2 -10916.684} C_VEL
LIN {X 0,Y 414.65,Z 478.195,A -85,B 0,C 180,E1 -10917.289,E2 -10917.289} C_VEL
LIN {X 0,Y 412.718,Z 464.644,A -85,B 0,C 180,E1 -10917.72,E2 -10917.72} C_VEL
LIN {X 0,Y 411.634,Z 451.22,A -85,B 0,C 180,E1 -10918.429,E2 -10918.429} C_VEL
LIN {X 0,Y 413.886,Z 424.952,A -85,B 0,C 180,E1 -10921.617,E2 -10921.617} C_VEL
LIN {X 0,Y 414.514,Z 417.157,A -85,B 0,C 180,E1 -10922.579,E2 -10922.579} C_VEL
LIN {X 0,Y 410.547,Z 402.548,A -85,B 0,C 180,E1 -10924.745,E2 -10924.745} C_VEL
LIN {X 0,Y 404.656,Z 382.707,A -85,B 0,C 180,E1 -10927.857,E2 -10927.857} C_VEL
LIN {X 0,Y 404.166,Z 380.936,A -85,B 0,C 180,E1 -10928.181,E2 -10928.181} C_VEL
LIN {X 0,Y 404.097,Z 380.775,A -85,B 0,C 180,E1 -10931.596,E2 -10931.596} C_VEL
LIN {X 0,Y 404.132,Z 380.772,A -85,B 0,C 180,E1 -10934.52,E2 -10934.52} C_VEL
LIN {X 0,Y 404.107,Z 380.74,A -85,B 0,C 180,E1 -10937.292,E2 -10937.292} C_VEL
LIN {X 0,Y 404.12,Z 380.763,A -85,B 0,C 180,E1 -10939.95,E2 -10939.95} C_VEL
LIN {X 0,Y 404.117,Z 380.75,A -85,B 0,C 180,E1 -10943.125,E2 -10943.125} C_VEL
LIN {X 0,Y 404.124,Z 380.743,A -85,B 0,C 180,E1 -10946.186,E2 -10946.186} C_VEL
LIN {X 0,Y 404.13,Z 380.768,A -85,B 0,C 180,E1 -10949.714,E2 -10949.714} C_VEL
LIN {X 0,Y 404.104,Z 380.771,A -85,B 0,C 180,E1 -10953.116,E2 -10953.116} C_VEL
LIN {X 0,Y 404.134,Z 380.762,A -85,B 0,C 180,E1 -10956.423,E2 -10956.423} C_VEL
LIN {X 0,Y 404.176,Z 380.752,A -85,B 0,C 180,E1 -10959.874,E2 -10959.874} C_VEL
LIN {X 0,Y 404.158,Z 380.764,A -85,B 0,C 180,E1 -10963.012,E2 -10963.012} C_VEL
LIN {X 0,Y 404.268,Z 380.753,A -85,B 0,C 180,E1 -10966.938,E2 -10966.938} C_VEL
LIN {X 0,Y 404.231,Z 380.745,A -85,B 0,C 180,E1 -10969.988,E2 -10969.988} C_VEL
LIN {X 0,Y 404.32,Z 380.745,A -85,B 0,C 180,E1 -10973.011,E2 -10973.011} C_VEL
LIN {X 0,Y 404.242,Z 380.741,A -85,B 0,C 180,E1 -10975.013,E2 -10975.013} C_VEL
LIN {X 0,Y 404.458,Z 380.726,A -85,B 0,C 180,E1 -10978.009,E2 -10978.009} C_VEL
LIN {X 0,Y 404.455,Z 380.716,A -85,B 0,C 180,E1 -10981.992,E2 -10981.992} C_VEL
LIN {X 0,Y 404.356,Z 380.728,A -85,B 0,C 180,E1 -10986.708,E2 -10986.708} C_VEL
LIN {X 0,Y 404.235,Z 380.754,A -85,B 0,C 180,E1 -10990.012,E2 -10990.012} C_VEL
LIN {X 0,Y 404.252,Z 380.751,A -85,B 0,C 180,E1 -10993.212,E2 -10993.212} C_VEL
LIN {X 0,Y 404.201,Z 380.749,A -85,B 0,C 180,E1 -10997.008,E2 -10997.008} C_VEL
LIN {X 0,Y 404.149,Z 380.761,A -85,B 0,C 180,E1 -11000.352,E2 -11000.352} C_VEL
LIN {X 0,Y 404.134,Z 380.767,A -85,B 0,C 180,E1 -11003.577,E2 -11003.577} C_VEL
LIN {X 0,Y 404.084,Z 380.776,A -85,B 0,C 180,E1 -11006.885,E2 -11006.885} C_VEL
LIN {X 0,Y 404.127,Z 380.767,A -85,B 0,C 180,E1 -11010.287,E2 -11010.287} C_VEL
LIN {X 0,Y 404.125,Z 380.77,A -85,B 0,C 180,E1 -11013.814,E2 -11013.814} C_VEL
LIN {X 0,Y 404.119,Z 380.745,A -85,B 0,C 180,E1 -11016.875,E2 -11016.875} C_VEL
LIN {X 0,Y 404.105,Z 380.773,A -85,B 0,C 180,E1 -11020.076,E2 -11020.076} C_VEL
LIN {X 0,Y 404.129,Z 380.75,A -85,B 0,C 180,E1 -11023.083,E2 -11023.083} C_VEL
LIN {X 0,Y 404.108,Z 380.761,A -85,B 0,C 180,E1 -11025.923,E2 -11025.923} C_VEL
LIN {X 0,Y 404.124,Z 380.759,A -85,B 0,C 180,E1 -11029.66,E2 -11029.66} C_VEL
LIN {X 0,Y 404.161,Z 381.033,A -85,B 0,C 180,E1 -11029.957,E2 -11029.957} C_VEL
LIN {X 0,Y 409.384,Z 396.274,A -85,B 0,C 180,E1 -11032.503,E2 -11032.503} C_VEL
LIN {X 0,Y 413.674,Z 410.307,A -85,B 0,C 180,E1 -11034.718,E2 -11034.718} C_VEL
LIN {X 0,Y 416.369,Z 420.681,A -85,B 0,C 180,E1 -11036.283,E2 -11036.283} C_VEL
LIN {X 0,Y 414.521,Z 448.449,A -85,B 0,C 180,E1 -11039.607,E2 -11039.607} C_VEL
LIN {X 0,Y 413.21,Z 471.624,A -85,B 0,C 180,E1 -11042.234,E2 -11042.234} C_VEL
LIN {X 0,Y 417.996,Z 501.985,A -85,B 0,C 180,E1 -11043.171,E2 -11043.171} C_VEL
LIN {X 0,Y 415.286,Z 639.806,A -85,B 0,C 180,E1 -11045.606,E2 -11045.606} C_VEL
LIN {X 0,Y 414.65,Z 655.621,A -85,B 0,C 180,E1 -11046.067,E2 -11046.067} C_VEL
LIN {X 0,Y 413.732,Z 669.889,A -85,B 0,C 180,E1 -11046.667,E2 -11046.667} C_VEL
LIN {X 0,Y 412.674,Z 684.185,A -85,B 0,C 180,E1 -11047.471,E2 -11047.471} C_VEL
LIN {X 0,Y 411.35,Z 697.982,A -85,B 0,C 180,E1 -11048.451,E2 -11048.451} C_VEL
LIN {X 0,Y 410.071,Z 710.647,A -85,B 0,C 180,E1 -11049.564,E2 -11049.564} C_VEL
LIN {X 0,Y 408.685,Z 723.425,A -85,B 0,C 180,E1 -11050.931,E2 -11050.931} C_VEL
LIN {X 0,Y 407.358,Z 735.007,A -85,B 0,C 180,E1 -11052.429,E2 -11052.429} C_VEL
LIN {X 0,Y 406.367,Z 743.482,A -85,B 0,C 180,E1 -11053.714,E2 -11053.714} C_VEL
LIN {X 0,Y 405.28,Z 747.313,A -85,B 0,C 180,E1 -11054.34,E2 -11054.34} C_VEL
LIN {X 0,Y 401.826,Z 753.291,A -85,B 0,C 180,E1 -11055.354,E2 -11055.354} C_VEL
LIN {X 0,Y 398.428,Z 758.779,A -85,B 0,C 180,E1 -11056.425,E2 -11056.425} C_VEL
LIN {X 0,Y 397.433,Z 761.858,A -85,B 0,C 180,E1 -11057.133,E2 -11057.133} C_VEL
LIN {X 0,Y 396.816,Z 767.952,A -85,B 0,C 180,E1 -11058.767,E2 -11058.767} C_VEL
LIN {X 0,Y 396.274,Z 774.204,A -85,B 0,C 180,E1 -11060.817,E2 -11060.817} C_VEL
LIN {X 0,Y 395.926,Z 779.036,A -85,B 0,C 180,E1 -11062.864,E2 -11062.864} C_VEL
LIN {X 0,Y 395.796,Z 782.578,A -85,B 0,C 180,E1 -11064.908,E2 -11064.908} C_VEL
LIN {X 0,Y 395.68,Z 784.92,A -85,B 0,C 180,E1 -11066.947,E2 -11066.947} C_VEL
LIN {X 0,Y 395.754,Z 786.113,A -85,B 0,C 180,E1 -11068.984,E2 -11068.984} C_VEL
LIN {X 0,Y 395.755,Z 786.128,A -85,B 0,C 180,E1 -11071.019,E2 -11071.019} C_VEL
LIN {X 0,Y 395.681,Z 784.995,A -85,B 0,C 180,E1 -11073.056,E2 -11073.056} C_VEL
LIN {X 0,Y 395.805,Z 782.712,A -85,B 0,C 180,E1 -11075.095,E2 -11075.095} C_VEL
LIN {X 0,Y 395.993,Z 779.224,A -85,B 0,C 180,E1 -11077.138,E2 -11077.138} C_VEL
LIN {X 0,Y 396.269,Z 774.453,A -85,B 0,C 180,E1 -11079.186,E2 -11079.186} C_VEL
LIN {X 0,Y 396.802,Z 768.276,A -85,B 0,C 180,E1 -11081.236,E2 -11081.236} C_VEL
LIN {X 0,Y 397.454,Z 761.605,A -85,B 0,C 180,E1 -11083.031,E2 -11083.031} C_VEL
LIN {X 0,Y 398.308,Z 753.517,A -85,B 0,C 180,E1 -11084.825,E2 -11084.825} C_VEL
LIN {X 0,Y 399.47,Z 743.805,A -85,B 0,C 180,E1 -11086.614,E2 -11086.614} C_VEL
LIN {X 0,Y 400.735,Z 733.856,A -85,B 0,C 180,E1 -11088.139,E2 -11088.139} C_VEL
LIN {X 0,Y 402.071,Z 722.039,A -85,B 0,C 180,E1 -11089.664,E2 -11089.664} C_VEL
LIN {X 0,Y 403.479,Z 710.243,A -85,B 0,C 180,E1 -11090.922,E2 -11090.922} C_VEL
LIN {X 0,Y 404.787,Z 697.501,A -85,B 0,C 180,E1 -11092.054,E2 -11092.054} C_VEL
LIN {X 0,Y 406.19,Z 683.581,A -85,B 0,C 180,E1 -11093.047,E2 -11093.047} C_VEL
LIN {X 0,Y 407.234,Z 669.555,A -85,B 0,C 180,E1 -11093.841,E2 -11093.841} C_VEL
LIN {X 0,Y 408.18,Z 655.332,A -85,B 0,C 180,E1 -11094.443,E2 -11094.443} C_VEL
LIN {X 0,Y 408.867,Z 639.429,A -85,B 0,C 180,E1 -11094.907,E2 -11094.907} C_VEL
LIN {X 0,Y 411.698,Z 502.447,A -85,B 0,C 180,E1 -11097.36,E2 -11097.36} C_VEL
LIN {X 0,Y 406.729,Z 471.427,A -85,B 0,C 180,E1 -11098.359,E2 -11098.359} C_VEL
LIN {X 0,Y 408.101,Z 448.837,A -85,B 0,C 180,E1 -11100.949,E2 -11100.949} C_VEL
LIN {X 0,Y 409.9,Z 422.904,A -85,B 0,C 180,E1 -11104.084,E2 -11104.084} C_VEL
LIN {X 0,Y 405.712,Z 407.716,A -85,B 0,C 180,E1 -11106.443,E2 -11106.443} C_VEL
LIN {X 0,Y 400.568,Z 391.587,A -85,B 0,C 180,E1 -11109.071,E2 -11109.071} C_VEL
LIN {X 0,Y 397.122,Z 381.907,A -85,B 0,C 180,E1 -11110.77,E2 -11110.77} C_VEL
LIN {X 0,Y 397.045,Z 381.655,A -85,B 0,C 180,E1 -11113.658,E2 -11113.658} C_VEL
LIN {X 0,Y 397.087,Z 381.635,A -85,B 0,C 180,E1 -11116.525,E2 -11116.525} C_VEL
